// TwinCAT 3 PLC project PulsePower_PLC
// ProgramVersion: 3.1.4023.0
// libraries:
//   Tc2_BACnetRev12, * (Beckhoff Automation GmbH)
//   Tc2_DataExchange, * (Beckhoff Automation GmbH)
//   Tc2_Math, * (Beckhoff Automation GmbH)
//   Tc2_NC, * (Beckhoff Automation GmbH)
//   Tc2_Standard, * (Beckhoff Automation GmbH)
//   Tc2_System, * (Beckhoff Automation GmbH)
//   Tc3_EventLogger, * (Beckhoff Automation GmbH)
//   Tc3_Module, * (Beckhoff Automation GmbH)
// project tree:
//   DUTs/ E_Command.TcDUT, E_PulseState.TcDUT, E_Status.TcDUT, ST_Alarm_Base.TcDUT (not stored), ST_Charger_Base.TcDUT, ST_ChargeTime.TcDUT (not stored), ST_Control.TcDUT, ST_Echo_MCP.TcDUT, ST_Echo_Section.TcDUT, ST_FieldDevices_Base.TcDUT, ST_FieldDevices_Form.TcDUT (not stored), ST_InstrumentReading.TcDUT, ST_Recipe.TcDUT, ST_RelayFaults_Base.TcDUT (not stored), ST_RelayFaults_Form.TcDUT (not stored), ST_Section_Base.TcDUT (not stored), ST_Setpoints_Base.TcDUT (not stored), ST_Trip_Base.TcDUT (not stored), ST_VoltageFeedback.TcDUT (not stored)
//   GVLs/ Alarms_DB.TcGVL, ChargeTime_DB.TcGVL (not stored), Command.TcGVL (not stored), EngVal.TcGVL, GVL.TcGVL (not stored), Recipe.TcGVL, Setpoints.TcGVL, TxMainPLC.TcGVL, HMI_DB.TcGVL, Input.TcGVL, InstrumentReading.TcGVL, LCP.TcGVL (not stored), MCP_IO.TcGVL, Output.TcGVL, Permissives_DB.TcGVL, Trips_DB.TcGVL
//   / PlcTask.TcTTO
//   POUs/ ADC_10V.TcPOU (not stored), ADC_5V.TcPOU (not stored), Alarms.TcPOU, Alarms_FB.TcPOU (not stored), Alias.TcPOU, AnalogConversion.TcPOU, AQ.TcPOU (not stored), ChargeTime.TcPOU, Communication.TcPOU, Dump_FB.TcPOU, Heartbeat.TcPOU (not stored), Heartbeat_1.TcPOU, HMI.TcPOU, LCA_CAL.TcPOU (not stored), MAIN.TcPOU, Norm_x.TcPOU (not stored), Permissives.TcPOU, PWMO.TcPOU (not stored), Sequence.TcPOU, Trips.TcPOU
// real-time tasks:
//   TASK PlcTask: cycle T#2ms, priority 20, ADS port 350
// I/O:
//   DEVICE Device 3 (EtherCAT) (disabled), AmsNetId 5.107.141.148.4.1
//     Term 23 (EK1101) [EK1101 EtherCAT Coupler (2A E-Bus, ID switch)]
//       Term 24 (EL2008) [EL2008 8Ch. Dig. Output 24V, 0.5A]
//       Term 25 (EL2008) [EL2008 8Ch. Dig. Output 24V, 0.5A]
//       Term 26 (EL3068) [EL3068 8Ch. Ana. Input 0-10V]
//       Term 27 (EL3068) [EL3068 8Ch. Ana. Input 0-10V]
//       Term 28 (EL4008) [EL4008 8K. Ana. Ausgang 0-10V, 12bit]
//       Term 29 (EL2008) [EL2008 8Ch. Dig. Output 24V, 0.5A]
//       Term 30 (EL4008) [EL4008 8K. Ana. Ausgang 0-10V, 12bit]
//       Term 18 (EL9011) [EL9011 End Terminal]
//   DEVICE Device 2 (EtherCAT) (disabled), AmsNetId 5.107.141.148.3.1
//     Term 4 (EK1200) [EK1200-5000 EtherCAT Power supply (2A E-Bus)]
//       Term 2 (EL1008) [EL1008 8Ch. Dig. Input 24V, 3ms]
//       Term 3 (EL1008) [EL1008 8Ch. Dig. Input 24V, 3ms]
//       Term 4 (EL1008) [EL1008 8Ch. Dig. Input 24V, 3ms]
//       Term 5 (EL1008) [EL1008 8Ch. Dig. Input 24V, 3ms]
//       Term 6 (EL1008) [EL1008 8Ch. Dig. Input 24V, 3ms]
//       Term 7 (EL1008) [EL1008 8Ch. Dig. Input 24V, 3ms]
//       Term 11 (EL1008) [EL1008 8Ch. Dig. Input 24V, 3ms]
//       Term 12 (EL1008) [EL1008 8Ch. Dig. Input 24V, 3ms]
//       Term 13 (EL1008) [EL1008 8Ch. Dig. Input 24V, 3ms]
//       Term 14 (EL6695) [EL6695 EtherCAT Bridge terminal (Primary)]
//       Term 15 (EK1561) [EK1561 1 port EtherCAT junction (POF)]
//       Term 16 (EL9011) [EL9011 End Terminal]
// variable links:
//   PulsePower_PLC/PulsePower_PLC Instance <-> Device 2 (EtherCAT)/Term 4 (EK1200)/Term 11 (EL1008)
//     PlcTask Inputs/Input.R1_07_00 <-> Channel 1/Input
//     PlcTask Inputs/Input.R1_07_01 <-> Channel 2/Input
//     PlcTask Inputs/Input.R1_07_02 <-> Channel 3/Input
//     PlcTask Inputs/Input.R1_07_03 <-> Channel 4/Input
//     PlcTask Inputs/Input.R1_07_04 <-> Channel 5/Input
//     PlcTask Inputs/Input.R1_07_05 <-> Channel 6/Input
//     PlcTask Inputs/Input.R1_07_06 <-> Channel 7/Input
//     PlcTask Inputs/Input.R1_07_07 <-> Channel 8/Input
//   PulsePower_PLC/PulsePower_PLC Instance <-> Device 2 (EtherCAT)/Term 4 (EK1200)/Term 12 (EL1008)
//     PlcTask Inputs/Input.R1_08_00 <-> Channel 1/Input
//     PlcTask Inputs/Input.R1_08_01 <-> Channel 2/Input
//     PlcTask Inputs/Input.R1_08_02 <-> Channel 3/Input
//     PlcTask Inputs/Input.R1_08_03 <-> Channel 4/Input
//     PlcTask Inputs/Input.R1_08_04 <-> Channel 5/Input
//     PlcTask Inputs/Input.R1_08_05 <-> Channel 6/Input
//     PlcTask Inputs/Input.R1_08_06 <-> Channel 7/Input
//     PlcTask Inputs/Input.R1_08_07 <-> Channel 8/Input
//   PulsePower_PLC/PulsePower_PLC Instance <-> Device 2 (EtherCAT)/Term 4 (EK1200)/Term 13 (EL1008)
//     PlcTask Inputs/Input.R1_09_00 <-> Channel 1/Input
//     PlcTask Inputs/Input.R1_09_01 <-> Channel 2/Input
//     PlcTask Inputs/Input.R1_09_02 <-> Channel 3/Input
//     PlcTask Inputs/Input.R1_09_03 <-> Channel 4/Input
//     PlcTask Inputs/Input.R1_09_04 <-> Channel 5/Input
//     PlcTask Inputs/Input.R1_09_05 <-> Channel 6/Input
//     PlcTask Inputs/Input.R1_09_06 <-> Channel 7/Input
//     PlcTask Inputs/Input.R1_09_07 <-> Channel 8/Input
//   PulsePower_PLC/PulsePower_PLC Instance <-> Device 2 (EtherCAT)/Term 4 (EK1200)/Term 2 (EL1008)
//     PlcTask Inputs/Input.R1_01_00 <-> Channel 1/Input
//     PlcTask Inputs/Input.R1_01_01 <-> Channel 2/Input
//     PlcTask Inputs/Input.R1_01_02 <-> Channel 3/Input
//     PlcTask Inputs/Input.R1_01_03 <-> Channel 4/Input
//     PlcTask Inputs/Input.R1_01_04 <-> Channel 5/Input
//     PlcTask Inputs/Input.R1_01_05 <-> Channel 6/Input
//     PlcTask Inputs/Input.R1_01_06 <-> Channel 7/Input
//     PlcTask Inputs/Input.R1_01_07 <-> Channel 8/Input
//   PulsePower_PLC/PulsePower_PLC Instance <-> Device 2 (EtherCAT)/Term 4 (EK1200)/Term 3 (EL1008)
//     PlcTask Inputs/Input.R1_02_00 <-> Channel 1/Input
//     PlcTask Inputs/Input.R1_02_01 <-> Channel 2/Input
//     PlcTask Inputs/Input.R1_02_02 <-> Channel 3/Input
//     PlcTask Inputs/Input.R1_02_03 <-> Channel 4/Input
//     PlcTask Inputs/Input.R1_02_04 <-> Channel 5/Input
//     PlcTask Inputs/Input.R1_02_05 <-> Channel 6/Input
//     PlcTask Inputs/Input.R1_02_06 <-> Channel 7/Input
//     PlcTask Inputs/Input.R1_02_07 <-> Channel 8/Input
//   PulsePower_PLC/PulsePower_PLC Instance <-> Device 2 (EtherCAT)/Term 4 (EK1200)/Term 4 (EL1008)
//     PlcTask Inputs/Input.R1_03_00 <-> Channel 1/Input
//     PlcTask Inputs/Input.R1_03_01 <-> Channel 2/Input
//     PlcTask Inputs/Input.R1_03_02 <-> Channel 3/Input
//     PlcTask Inputs/Input.R1_03_03 <-> Channel 4/Input
//     PlcTask Inputs/Input.R1_03_04 <-> Channel 5/Input
//     PlcTask Inputs/Input.R1_03_05 <-> Channel 6/Input
//     PlcTask Inputs/Input.R1_03_06 <-> Channel 7/Input
//     PlcTask Inputs/Input.R1_03_07 <-> Channel 8/Input
//   PulsePower_PLC/PulsePower_PLC Instance <-> Device 2 (EtherCAT)/Term 4 (EK1200)/Term 5 (EL1008)
//     PlcTask Inputs/Input.R1_04_00 <-> Channel 1/Input
//     PlcTask Inputs/Input.R1_04_01 <-> Channel 2/Input
//     PlcTask Inputs/Input.R1_04_02 <-> Channel 3/Input
//     PlcTask Inputs/Input.R1_04_03 <-> Channel 4/Input
//     PlcTask Inputs/Input.R1_04_04 <-> Channel 5/Input
//     PlcTask Inputs/Input.R1_04_05 <-> Channel 6/Input
//     PlcTask Inputs/Input.R1_04_06 <-> Channel 7/Input
//     PlcTask Inputs/Input.R1_04_07 <-> Channel 8/Input
//   PulsePower_PLC/PulsePower_PLC Instance <-> Device 2 (EtherCAT)/Term 4 (EK1200)/Term 6 (EL1008)
//     PlcTask Inputs/Input.R1_05_00 <-> Channel 1/Input
//     PlcTask Inputs/Input.R1_05_01 <-> Channel 2/Input
//     PlcTask Inputs/Input.R1_05_02 <-> Channel 3/Input
//     PlcTask Inputs/Input.R1_05_03 <-> Channel 4/Input
//     PlcTask Inputs/Input.R1_05_04 <-> Channel 5/Input
//     PlcTask Inputs/Input.R1_05_05 <-> Channel 6/Input
//     PlcTask Inputs/Input.R1_05_06 <-> Channel 7/Input
//     PlcTask Inputs/Input.R1_05_07 <-> Channel 8/Input
//   PulsePower_PLC/PulsePower_PLC Instance <-> Device 2 (EtherCAT)/Term 4 (EK1200)/Term 7 (EL1008)
//     PlcTask Inputs/Input.R1_06_00 <-> Channel 1/Input
//     PlcTask Inputs/Input.R1_06_01 <-> Channel 2/Input
//     PlcTask Inputs/Input.R1_06_02 <-> Channel 3/Input
//     PlcTask Inputs/Input.R1_06_03 <-> Channel 4/Input
//     PlcTask Inputs/Input.R1_06_04 <-> Channel 5/Input
//     PlcTask Inputs/Input.R1_06_05 <-> Channel 6/Input
//     PlcTask Inputs/Input.R1_06_06 <-> Channel 7/Input
//     PlcTask Inputs/Input.R1_06_07 <-> Channel 8/Input
//   PulsePower_PLC/PulsePower_PLC Instance <-> Device 3 (EtherCAT)/Term 23 (EK1101)/Term 24 (EL2008)
//     PlcTask Outputs/Output.R2_01_00 <-> Channel 1/Output
//     PlcTask Outputs/Output.R2_01_01 <-> Channel 2/Output
//     PlcTask Outputs/Output.R2_01_02 <-> Channel 3/Output
//     PlcTask Outputs/Output.R2_01_03 <-> Channel 4/Output
//     PlcTask Outputs/Output.R2_01_04 <-> Channel 5/Output
//     PlcTask Outputs/Output.R2_01_05 <-> Channel 6/Output
//     PlcTask Outputs/Output.R2_01_06 <-> Channel 7/Output
//     PlcTask Outputs/Output.R2_01_07 <-> Channel 8/Output
//   PulsePower_PLC/PulsePower_PLC Instance <-> Device 3 (EtherCAT)/Term 23 (EK1101)/Term 25 (EL2008)
//     PlcTask Outputs/Output.R2_02_00 <-> Channel 1/Output
//     PlcTask Outputs/Output.R2_02_01 <-> Channel 2/Output
//     PlcTask Outputs/Output.R2_02_02 <-> Channel 3/Output
//     PlcTask Outputs/Output.R2_02_03 <-> Channel 4/Output
//     PlcTask Outputs/Output.R2_02_04 <-> Channel 5/Output
//     PlcTask Outputs/Output.R2_02_05 <-> Channel 6/Output
//     PlcTask Outputs/Output.R2_02_06 <-> Channel 7/Output
//     PlcTask Outputs/Output.R2_02_07 <-> Channel 8/Output
//   PulsePower_PLC/PulsePower_PLC Instance <-> Device 3 (EtherCAT)/Term 23 (EK1101)/Term 26 (EL3068)
//     PlcTask Inputs/Input.R2_03_00 <-> AI Standard Channel 1/Value
//     PlcTask Inputs/Input.R2_03_01 <-> AI Standard Channel 2/Value
//     PlcTask Inputs/Input.R2_03_02 <-> AI Standard Channel 3/Value
//     PlcTask Inputs/Input.R2_03_03 <-> AI Standard Channel 4/Value
//     PlcTask Inputs/Input.R2_03_04 <-> AI Standard Channel 5/Value
//     PlcTask Inputs/Input.R2_03_05 <-> AI Standard Channel 6/Value
//     PlcTask Inputs/Input.R2_03_06 <-> AI Standard Channel 7/Value
//     PlcTask Inputs/Input.R2_03_07 <-> AI Standard Channel 8/Value
//     PlcTask Inputs/Input.R2_03_00_Status <-> AI Standard Channel 1/Status
//     PlcTask Inputs/Input.R2_03_01_Status <-> AI Standard Channel 2/Status
//     PlcTask Inputs/Input.R2_03_02_Status <-> AI Standard Channel 3/Status
//     PlcTask Inputs/Input.R2_03_03_Status <-> AI Standard Channel 4/Status
//     PlcTask Inputs/Input.R2_03_04_Status <-> AI Standard Channel 5/Status
//     PlcTask Inputs/Input.R2_03_05_Status <-> AI Standard Channel 6/Status
//     PlcTask Inputs/Input.R2_03_06_Status <-> AI Standard Channel 7/Status
//     PlcTask Inputs/Input.R2_03_07_Status <-> AI Standard Channel 8/Status
//   PulsePower_PLC/PulsePower_PLC Instance <-> Device 3 (EtherCAT)/Term 23 (EK1101)/Term 27 (EL3068)
//     PlcTask Inputs/Input.R2_04_00 <-> AI Standard Channel 1/Value
//     PlcTask Inputs/Input.R2_04_01 <-> AI Standard Channel 2/Value
//     PlcTask Inputs/Input.R2_04_02 <-> AI Standard Channel 3/Value
//     PlcTask Inputs/Input.R2_04_03 <-> AI Standard Channel 4/Value
//     PlcTask Inputs/Input.R2_04_04 <-> AI Standard Channel 5/Value
//     PlcTask Inputs/Input.R2_04_05 <-> AI Standard Channel 6/Value
//     PlcTask Inputs/Input.R2_04_06 <-> AI Standard Channel 7/Value
//     PlcTask Inputs/Input.R2_04_07 <-> AI Standard Channel 8/Value
//     PlcTask Inputs/Input.R2_04_00_Status <-> AI Standard Channel 1/Status
//     PlcTask Inputs/Input.R2_04_01_Status <-> AI Standard Channel 2/Status
//     PlcTask Inputs/Input.R2_04_02_Status <-> AI Standard Channel 3/Status
//     PlcTask Inputs/Input.R2_04_03_Status <-> AI Standard Channel 4/Status
//     PlcTask Inputs/Input.R2_04_04_Status <-> AI Standard Channel 5/Status
//     PlcTask Inputs/Input.R2_04_05_Status <-> AI Standard Channel 6/Status
//     PlcTask Inputs/Input.R2_04_06_Status <-> AI Standard Channel 7/Status
//     PlcTask Inputs/Input.R2_04_07_Status <-> AI Standard Channel 8/Status
//   PulsePower_PLC/PulsePower_PLC Instance <-> Device 3 (EtherCAT)/Term 23 (EK1101)/Term 28 (EL4008)
//     PlcTask Outputs/Output.R2_05_00 <-> AO Outputs Channel 1/Analog output
//     PlcTask Outputs/Output.R2_05_01 <-> AO Outputs Channel 2/Analog output
//     PlcTask Outputs/Output.R2_05_02 <-> AO Outputs Channel 3/Analog output
//     PlcTask Outputs/Output.R2_05_03 <-> AO Outputs Channel 4/Analog output
//     PlcTask Outputs/Output.R2_05_04 <-> AO Outputs Channel 5/Analog output
//     PlcTask Outputs/Output.R2_05_05 <-> AO Outputs Channel 6/Analog output
//     PlcTask Outputs/Output.R2_05_06 <-> AO Outputs Channel 7/Analog output
//     PlcTask Outputs/Output.R2_05_07 <-> AO Outputs Channel 8/Analog output
//   PulsePower_PLC/PulsePower_PLC Instance <-> Device 3 (EtherCAT)/Term 23 (EK1101)/Term 29 (EL2008)
//     PlcTask Outputs/Output.R2_06_00 <-> Channel 1/Output
//     PlcTask Outputs/Output.R2_06_01 <-> Channel 2/Output
//     PlcTask Outputs/Output.R2_06_02 <-> Channel 3/Output
//     PlcTask Outputs/Output.R2_06_03 <-> Channel 4/Output
//     PlcTask Outputs/Output.R2_06_04 <-> Channel 5/Output
//     PlcTask Outputs/Output.R2_06_05 <-> Channel 6/Output
//     PlcTask Outputs/Output.R2_06_06 <-> Channel 7/Output
//     PlcTask Outputs/Output.R2_06_07 <-> Channel 8/Output
//   PulsePower_PLC/PulsePower_PLC Instance <-> Device 3 (EtherCAT)/Term 23 (EK1101)/Term 30 (EL4008)
//     PlcTask Outputs/Output.R2_07_00 <-> AO Outputs Channel 1/Analog output
//     PlcTask Outputs/Output.R2_07_01 <-> AO Outputs Channel 2/Analog output
//     PlcTask Outputs/Output.R2_07_02 <-> AO Outputs Channel 3/Analog output
//     PlcTask Outputs/Output.R2_07_03 <-> AO Outputs Channel 4/Analog output
//     PlcTask Outputs/Output.R2_07_04 <-> AO Outputs Channel 5/Analog output
//     PlcTask Outputs/Output.R2_07_05 <-> AO Outputs Channel 6/Analog output
//     PlcTask Outputs/Output.R2_07_06 <-> AO Outputs Channel 7/Analog output
//     PlcTask Outputs/Output.R2_07_07 <-> AO Outputs Channel 8/Analog output

CONFIGURATION PulsePower_PLC
    RESOURCE PLC ON TwinCAT3
        TASK PlcTask(INTERVAL := T#2ms, PRIORITY := 20);
        PROGRAM MAIN WITH PlcTask : MAIN;
        PROGRAM Heartbeat WITH PlcTask : Heartbeat;
        PROGRAM Heartbeat_1 WITH PlcTask : Heartbeat_1;
    END_RESOURCE
END_CONFIGURATION

// ---- DUTs/E_Command.TcDUT
{attribute 'qualified_only'}
{attribute 'strict'}
{attribute 'to_string'}
//Command from Master PLC (screenroom)
TYPE E_Command :
(
	//Requested PP State
	IDLE		 	:= 0, 
	CHARGE			:= 1, 
	DISCONNECT		:= 2,
	DUMP			:= 3, 
	ABORT			:= 4
);
END_TYPE

// ---- DUTs/E_PulseState.TcDUT
{attribute 'qualified_only'}
{attribute 'strict'}
TYPE E_PulseState :
(
	SAFE			:= 0, //IDLE
	CHARGING		:= 1, //Charge
	CHARGECOMPLETE	:= 2, //EOC
	DISCONNECTING	:= 3, //Disconnect
	DUMPING			:= 4, 
	ABORT			:= 5,
	TRIPPED			:= 6,
	LOCALMODE		:= 7	
);
END_TYPE

// ---- DUTs/E_Status.TcDUT
{attribute 'qualified_only'}
{attribute 'strict'}
{attribute 'to_string'}
TYPE E_Status :
(
	//Actual Pulse Power State
	SAFE			:= 0, //IDLE
	CHARGING		:= 1, //Charge
	CHARGECOMPLETE	:= 2, //EOC
	DISCONNECTING	:= 3, //Disconnect
	DISCONNECTED	:= 4,
	DUMPING			:= 5, 
	ABORT			:= 6,	
	TRIPPED			:= 7,
	LOCAL_MODE		:= 8
) ;
END_TYPE

// ---- DUTs/ST_Charger_Base.TcDUT
TYPE ST_Charger_Base :
STRUCT
	//DI
	inhibited 		: BOOL;
	EndOfCharge 	: BOOL;
	HV_isON			: BOOL;
	OverTemp		: BOOL;
	InterlockOpen	: BOOL;
	LoadFaulted		: BOOL;
	SummaryFaulted	: BOOL;
	
	//DQ
	inhibit			: BOOL;
	HV_ON			: BOOL;
	
	//AI
	voltageFeedback_raw 	: INT;
	voltageFeedback_norm 	: REAL;
	voltageFeedback			: REAL;
	
	currentFeedback_raw 	: INT;
	currentFeedback_norm	: REAL;
	currentFeedback			: REAL;
	
	//AQ
	voltageSP_norm	: REAL;
	voltageSP		: DINT;
	voltageSP_raw	: INT; // setpoint output to field device.
	
	//Internal
	ChargerType_50kV : BOOL;
	ChargerType_12kV : BOOL;
	LossInhibit		 : BOOL;
	LossHVON		 : BOOL;
	LossInhibitTON	 : TON;
	LossHVON_TON	 : TON;
	
	ChargeTime		: ST_ChargeTime;
END_STRUCT
END_TYPE

// ---- DUTs/ST_Control.TcDUT
TYPE ST_Control :
STRUCT
	ClearAllFaults : BOOL;
END_STRUCT
END_TYPE

// ---- DUTs/ST_Echo_MCP.TcDUT
TYPE ST_Echo_MCP :
STRUCT
	VoltageFeedback : REAL;
	CurrentFeedback : REAL;
	TDKLoad			: ST_ChargeTime;
	
END_STRUCT
END_TYPE

// ---- DUTs/ST_Echo_Section.TcDUT
TYPE ST_Echo_Section :
STRUCT
	PeakCap : ARRAY[1..10] OF ST_InstrumentReading;
	SustCap : ARRAY[1..2] OF ST_InstrumentReading;
	FormCap : ARRAY[1..12] OF ST_InstrumentReading;
	FormTrigVoltage		: REAL;
	PreFormTrigVoltage  : REAL;
	PreFormCapVoltage  : REAL;
END_STRUCT
END_TYPE

// ---- DUTs/ST_FieldDevices_Base.TcDUT
TYPE ST_FieldDevices_Base :
STRUCT
	Cap : ARRAY [1..12] OF ST_InstrumentReading;
	
	ChargeRelay1_close		:BOOL;
	ChargeRelay2_close		:BOOL;
	
	ShortContact1_close		:BOOL;
	UnshortContact1_close 	:BOOL;
	ShortContact1Engaged	:BOOL;
	ShortContact1unknown	:BOOL;
	
	ShortContact2_close		:BOOL;
	UnshortContact2_close 	:BOOL;
	ShortContact2Engaged	:BOOL;
	ShortContact2unknown	:BOOL;
	
	DumpRelay1_close		:BOOL;
	DumpRelay2_close		:BOOL;
	
	CloseChargeRelay1		:BOOL;
	CloseChargeRelay2		:BOOL;
	OpenDumpRelay1			:BOOL;
	OpenDumpRelay2			:BOOL;
	
	//Bank					: ST_ChargeTime;

END_STRUCT
END_TYPE

// ---- DUTs/ST_InstrumentReading.TcDUT
TYPE ST_InstrumentReading :
STRUCT
	
	(*CH00 : REAL;
	CH01 : REAL;
	CH02 : REAL;
	CH03 : REAL;
	CH04 : REAL;
	CH05 : REAL;
	CH06 : REAL;
	CH07 : REAL;
	R2_01_CH02 : REAL;
	R2_01_CH03 : REAL;
	R2_01_CH04 : REAL;
	R2_01_CH05 : REAL;
	R2_01_CH06 : REAL;
	R2_01_CH07 : REAL;*)
	voltageFeedback_raw		: INT;
	voltageFeedback_Norm 	: REAL;
	voltageFeedback 		: REAL;
	currentFeedback_raw		: INT;
	currentFeedback_Norm 	: REAL;
	currentFeedback 		: REAL;
	
	CapDischaged			: BOOL;
	CapFullyCharged			: BOOL;
END_STRUCT
END_TYPE

// ---- DUTs/ST_Recipe.TcDUT
TYPE ST_Recipe :
STRUCT
	RequiredChargedV : REAL := 10; //DINT;
END_STRUCT
END_TYPE

// ---- GVLs/Alarms_DB.TcGVL
{attribute 'qualified_only'}
VAR_GLOBAL
	MCP	: ST_Alarm_Base;
	Section1 : ST_Alarm_Base;
	Section2 : ST_Alarm_Base;
	Section3 : ST_Alarm_Base;
	Section4 : ST_Alarm_Base;
	
	AlarmWord5  : ST_Alarm_Base;
	AlarmWord6  : ST_Alarm_Base;
	AlarmWord7  : ST_Alarm_Base;
	AlarmWord8  : ST_Alarm_Base;
	AlarmWord9  : ST_Alarm_Base;
	//AlarmWord11 : ST_Alarm_Base;
	//AlarmWord12 : ST_Alarm_Base;
	//AlarmWord13 : ST_Alarm_Base;
	//AlarmWord14 : ST_Alarm_Base;
	//AlarmWord15 : ST_Alarm_Base;
END_VAR

// ---- GVLs/EngVal.TcGVL
{attribute 'qualified_only'}
VAR_GLOBAL
	Max_50kVChargerVoltage : REAL := 50000; //50kV
	Min_50kVChargerVoltage : REAL := 0;
	
	Max_50kVChargerCurrent : REAL := 0.18; //total peak charge current is 0.18A
	Min_50kVChargerCurrent : REAL := 0;
	
	Max_12kVChargerVoltage : REAL := 12000; //12kV
	Min_12kVChargerVoltage : REAL := 0;
	
	Max_12kVChargerCurrent : REAL := 0.75; //total peak charge current is 0.75A
	Min_12kVChargerCurrent : REAL := 0;
	
	Max_GLS1_ChargerV	   : REAL := 50000; //form trigger
	Max_GLS2_ChargerV	   : REAL := 50000; // preform trigger
	Max_GLS3_ChargerV	   : REAL := 30000; // preform cap charger
	
	Max_CapVoltage			: REAL := 32000;  //assuming 32kV cap....  
	Min_CapVoltage			: REAL := 0;
	
	ULimit_PeakCapRequiredV	: REAL := 10000; //10kV veto
	LLimit_PeakCapRequiredV	: REAL := -2000; //-2kV
	ULimit_SustCapRequiredV	: REAL := 12000; //12kv veto
	LLimit_SustCapRequiredV	: REAL := -2000; //-2kv
	ULimit_FormCapRequiredV : REAL := 35000;
	LLimit_FormCapRequiredV : REAL := 0;
	
	ULimit_PreFormCapRequiredV : REAL := 30000;
	LLimit_PreFormCapRequiredV : REAL := 0;
		
END_VAR

// ---- GVLs/Recipe.TcGVL
{attribute 'qualified_only'}
VAR_GLOBAL
	TDKLoad : ARRAY [1..8] OF ST_Recipe;
	GLSLoad : ST_Recipe;
	GLS1_VSP : REAL := 50; //DINT;
	GLS2_VSP : REAL := 50; //DINT;
END_VAR

// ---- GVLs/Setpoints.TcGVL
{attribute 'qualified_only'}
VAR_GLOBAL
	TDKLoad : ARRAY [1..8] OF ST_Setpoints_Base;
	GLSLoad : ST_Setpoints_Base;
	GLS1_VSP : REAL := 50;
	GLS2_VSP : REAL := 50;
END_VAR

// ---- GVLs/TxMainPLC.TcGVL
{attribute 'qualified_only'}
VAR_GLOBAL
	Charger		: ARRAY[1..8] OF ST_Echo_MCP;
	GLSLoad		: ST_ChargeTime;
	Section 	: ARRAY[1..4] OF ST_Echo_Section;
	ChargeRunOutTime	: REAL;
	ChargingRunOutTime	: REAL;
END_VAR

// ---- GVLs/HMI_DB.TcGVL
{attribute 'qualified_only'}
VAR_GLOBAL PERSISTENT
	RemoteModeSelected 	: BOOL := TRUE;
	
	OpenAllDumpRlyPB	: BOOL;
	CloseAllChargeRlyPB	: BOOL;
	AbortPB				: BOOL;
	
	ChargerHVOFF_rlyDelayPT		: TIME := T#25MS;
	ChargerHVOFF_rlyDelayPT_INT	: INT := 25;
	
	HVONdelayPT					: TIME := T#250MS;
	HVONdelayPT_INT				: INT := 250;
	
	RunOutTMR_PT				: TIME := T#10S;
	RunOutTMR_PT_INT			: INT := 10;
	RunOutTMR_elapse			: INT;
	
	ChargingRunOutTMR_elapse	: INT;
	
	//admin bypasses
	SafetyOKBP					: BOOL;
	AllDumpRelaysOpenBP			: BOOL;
	InterlockPressureLossBP		: BOOL;
	AllChargeRelayCloseBP		: BOOL;
	NoFaultDetectedBP			: BOOL;
	//AllShortingSysRemovedBP		: BOOL;
	AlldcPSUokBP				: BOOL;
	LossHVsignalBP				: BOOL;
	
	//timeToChargeLoad 			: ARRAY [1..8] OF REAL;
	//GLSchargeTime	 			: ARRAY [1..3] OF REAL;
	TDKLoad 					: ARRAY [1..8] OF ST_Setpoints_Base; //or RETAIN
	GLSLoad	 					: ST_Setpoints_Base;
	
	(*PSratedV					: REAL := 50;
	RequiredChargeV				: REAL := 30;
	LoadCapacitance				: REAL := 600;
	wLCA						: BOOL := TRUE;
	NumOfCharger				: INT := 1;*)
END_VAR

VAR_GLOBAL
	LiftMachineGNDsw			: BOOL;
	//for startup run
	PeakChargerSP				: DINT;
	SustChargerSP				: DINT;
	FormChargerSP				: DINT;
	PreFormChargerSP			: DINT;
	FormTrigChargerSP			: DINT;
	PreFormTrigChargerSP		: DINT;
	
	OpenAllPeakDumpRlySW		: BOOL;
	OpenAllSustDumpRlySW		: BOOL;
	OpenAllFormDumpRlySW		: BOOL;
	OpenAllPreFormDumpRlySW		: BOOL;
	OpenFormTrigDumpRlySW		: BOOL;
	OpenPreFormTrigDumpRlySW	: BOOL;
	
	CloseAllPeakChargRlySW		: BOOL;
	CloseAllSustChargRlySW		: BOOL;
	CloseAllFormChargRlySW		: BOOL;
	CloseAllPreFormChargRlySW	: BOOL;
	CloseFormTrigChargeRlySW	: BOOL;
	ClosePreFormTrigChargeRlySW : BOOL;
	
	PeakHVONsw					: BOOL; //enable
	SustHVONsw					: BOOL; //enable
	FormHVONsw					: BOOL; //enable
	PreFormHVONsw				: BOOL;
	GLS1HVONsw					: BOOL;
	GLS2HVONsw					: BOOL;
	
	ResetPB_Local				: BOOL;
	
	(*PeakInhibitONsw				: BOOL;
	SustInhibitONsw				: BOOL;
	FormInhibitONsw				: BOOL;
	PreFormInhibitONsw			: BOOL;
	*)	
END_VAR

// ---- GVLs/Input.TcGVL
{attribute 'qualified_only'}
VAR_GLOBAL
//***MCP************************************************************************
	//EL1008 - DI1
	R1_01_00 AT	%I*: BOOL; //Master stop PB not pressed - black pb on mcp
	R1_01_01 AT	%I*: BOOL; //case Estop circuit okay (Rly1 (120vac)
	R1_01_02 AT %I*: BOOL; //Remote Mode Selected (NO)
	R1_01_03 AT %I*: BOOL; //MCP PSU1 DC OK
	R1_01_04 AT %I*: BOOL; //Machine Ground Relay Open (lifted) Opto Board
	R1_01_05 AT %I*: BOOL; //spare
	R1_01_06 AT %I*: BOOL; //spare
	R1_01_07 AT %I*: BOOL; //spare

	//EL1008 - DI2
	//TDK802 1
	R1_02_00 AT	%I*: BOOL; 
	R1_02_01 AT	%I*: BOOL;
	R1_02_02 AT %I*: BOOL; 
	R1_02_03 AT %I*: BOOL; 
	R1_02_04 AT %I*: BOOL; 
	R1_02_05 AT %I*: BOOL; 
	R1_02_06 AT %I*: BOOL; 
	R1_02_07 AT %I*: BOOL; //spare
	
	//EL1008 - DI3
	//TDK802 2
	R1_03_00 AT	%I*: BOOL; 
	R1_03_01 AT	%I*: BOOL;
	R1_03_02 AT %I*: BOOL; 
	R1_03_03 AT %I*: BOOL; 
	R1_03_04 AT %I*: BOOL; 
	R1_03_05 AT %I*: BOOL; 
	R1_03_06 AT %I*: BOOL; 
	R1_03_07 AT %I*: BOOL; //spare
		
	//EL1008 - DI4
	//TDK802 3
	R1_04_00 AT	%I*: BOOL; 
	R1_04_01 AT	%I*: BOOL;
	R1_04_02 AT %I*: BOOL; 
	R1_04_03 AT %I*: BOOL; 
	R1_04_04 AT %I*: BOOL; 
	R1_04_05 AT %I*: BOOL; 
	R1_04_06 AT %I*: BOOL; 
	R1_04_07 AT %I*: BOOL; //spare
	
	//EL1008 - DI5
	//TDK802 4
	R1_05_00 AT	%I*: BOOL; 
	R1_05_01 AT	%I*: BOOL;
	R1_05_02 AT %I*: BOOL; 
	R1_05_03 AT %I*: BOOL; 
	R1_05_04 AT %I*: BOOL; 
	R1_05_05 AT %I*: BOOL; 
	R1_05_06 AT %I*: BOOL; 
	R1_05_07 AT %I*: BOOL; //spare
	
	//EL1008 - DI6
	//TDK802 5
	R1_06_00 AT	%I*: BOOL; 
	R1_06_01 AT	%I*: BOOL;
	R1_06_02 AT %I*: BOOL; 
	R1_06_03 AT %I*: BOOL; 
	R1_06_04 AT %I*: BOOL; 
	R1_06_05 AT %I*: BOOL; 
	R1_06_06 AT %I*: BOOL; 
	R1_06_07 AT %I*: BOOL; //spare
	
	//EL1008 - DI7
	//TDK802 6
	R1_07_00 AT	%I*: BOOL; 
	R1_07_01 AT	%I*: BOOL;
	R1_07_02 AT %I*: BOOL; 
	R1_07_03 AT %I*: BOOL; 
	R1_07_04 AT %I*: BOOL; 
	R1_07_05 AT %I*: BOOL; 
	R1_07_06 AT %I*: BOOL; 
	R1_07_07 AT %I*: BOOL; //spare
	
	//EL1008 - DI8
	//TDK802 7
	R1_08_00 AT	%I*: BOOL; 
	R1_08_01 AT	%I*: BOOL;
	R1_08_02 AT %I*: BOOL; 
	R1_08_03 AT %I*: BOOL; 
	R1_08_04 AT %I*: BOOL; 
	R1_08_05 AT %I*: BOOL; 
	R1_08_06 AT %I*: BOOL; 
	R1_08_07 AT %I*: BOOL; //spare
	
	//EL1008 - DI9
	//TDK802 8
	R1_09_00 AT	%I*: BOOL; 
	R1_09_01 AT	%I*: BOOL;
	R1_09_02 AT %I*: BOOL; 
	R1_09_03 AT %I*: BOOL; 
	R1_09_04 AT %I*: BOOL; 
	R1_09_05 AT %I*: BOOL; 
	R1_09_06 AT %I*: BOOL; 
	R1_09_07 AT %I*: BOOL; //spare

//RACK 2
	//EL3068 - AI1
	R2_03_00 		AT %I*: INT;
	R2_03_00_Status AT %I*: WORD;

	R2_03_01 		AT %I*: INT;
	R2_03_01_Status AT %I*: WORD;

	R2_03_02 		AT %I*: INT;
	R2_03_02_Status AT %I*: WORD;

	R2_03_03 		AT %I*: INT;
	R2_03_03_Status AT %I*: WORD;

	R2_03_04 		AT %I*: INT;
	R2_03_04_Status AT %I*: WORD;

	R2_03_05 		AT %I*: INT;
	R2_03_05_Status AT %I*: WORD;

	R2_03_06 		AT %I*: INT;
	R2_03_06_Status AT %I*: WORD;

	R2_03_07 		AT %I*: INT;
	R2_03_07_Status AT %I*: WORD;


	//EL3068 - AI2
	R2_04_00 		AT %I*: INT;
	R2_04_00_Status AT %I*: WORD;

	R2_04_01 		AT %I*: INT;
	R2_04_01_Status AT %I*: WORD;

	R2_04_02 		AT %I*: INT;
	R2_04_02_Status AT %I*: WORD;

	R2_04_03 		AT %I*: INT;
	R2_04_03_Status AT %I*: WORD;

	R2_04_04 		AT %I*: INT;
	R2_04_04_Status AT %I*: WORD;

	R2_04_05 		AT %I*: INT;
	R2_04_05_Status AT %I*: WORD;

	R2_04_06 		AT %I*: INT;
	R2_04_06_Status AT %I*: WORD;

	R2_04_07 		AT %I*: INT;
	R2_04_07_Status AT %I*: WORD;

//***LCP1***BANK1 (Rack 3)********************************************************************
//EL3068 - AI1
	R3_01_00 		AT %I*: INT;
	R3_01_00_Status AT %I*: WORD;
	
	R3_01_01		AT %I*: INT;
	R3_01_01_Status AT %I*: WORD;
	
	R3_01_02 		AT %I*: INT;
	R3_01_02_Status AT %I*: WORD;
	
	R3_01_03 		AT %I*: INT;
	R3_01_03_Status AT %I*: WORD;
	
	R3_01_04 		AT %I*: INT;
	R3_01_04_Status AT %I*: WORD;
	
	R3_01_05 		AT %I*: INT;
	R3_01_05_Status AT %I*: WORD;
	
	R3_01_06 		AT %I*: INT;
	R3_01_06_Status AT %I*: WORD;
	
	R3_01_07 		AT %I*: INT;
	R3_01_07_Status AT %I*: WORD;
	
	//EL3068 - AI2
	R3_02_00 		AT %I*: INT;
	R3_02_00_Status AT %I*: WORD;
	
	R3_02_01		AT %I*: INT;
	R3_02_01_Status AT %I*: WORD;
	
	R3_02_02 		AT %I*: INT;
	R3_02_02_Status AT %I*: WORD;
	
	R3_02_03 		AT %I*: INT;
	R3_02_03_Status AT %I*: WORD;
	
	R3_02_04 		AT %I*: INT; //SPARE
	R3_02_04_Status AT %I*: WORD;
	
	R3_02_05 		AT %I*: INT; //SPARE
	R3_02_05_Status AT %I*: WORD;
	
	R3_02_06 		AT %I*: INT; //SPARE
	R3_02_06_Status AT %I*: WORD;
	
	R3_02_07 		AT %I*: INT; //SPARE
	R3_02_07_Status AT %I*: WORD;

//EL1008 - DI1
	R3_03_00 AT %I*: BOOL;
	R3_03_01 AT %I*: BOOL;
	R3_03_02 AT %I*: BOOL;
	R3_03_03 AT %I*: BOOL;
	R3_03_04 AT %I*: BOOL;
	R3_03_05 AT %I*: BOOL;
	R3_03_06 AT %I*: BOOL;
	R3_03_07 AT %I*: BOOL;
//EL1008 - DI2	
	R3_04_00 AT %I*: BOOL;
	R3_04_01 AT %I*: BOOL;
	R3_04_02 AT %I*: BOOL;
	R3_04_03 AT %I*: BOOL;
	R3_04_04 AT %I*: BOOL;
	R3_04_05 AT %I*: BOOL; 
	R3_04_06 AT %I*: BOOL; //SPARE
	R3_04_07 AT %I*: BOOL; //SPARE

//***LCP2***BANK2 (Rack 4)********************************************************************
//EL3068 - AI1
	R4_01_00 		AT %I*: INT;
	R4_01_00_Status AT %I*: WORD;
	
	R4_01_01		AT %I*: INT;
	R4_01_01_Status AT %I*: WORD;
	
	R4_01_02 		AT %I*: INT;
	R4_01_02_Status AT %I*: WORD;
	
	R4_01_03 		AT %I*: INT;
	R4_01_03_Status AT %I*: WORD;
	
	R4_01_04 		AT %I*: INT;
	R4_01_04_Status AT %I*: WORD;
	
	R4_01_05 		AT %I*: INT;
	R4_01_05_Status AT %I*: WORD;
	
	R4_01_06 		AT %I*: INT;
	R4_01_06_Status AT %I*: WORD;
	
	R4_01_07 		AT %I*: INT;
	R4_01_07_Status AT %I*: WORD;
	
	//EL3068 - AI2
	R4_02_00 		AT %I*: INT;
	R4_02_00_Status AT %I*: WORD;
	
	R4_02_01		AT %I*: INT;
	R4_02_01_Status AT %I*: WORD;
	
	R4_02_02 		AT %I*: INT;
	R4_02_02_Status AT %I*: WORD;
	
	R4_02_03 		AT %I*: INT;
	R4_02_03_Status AT %I*: WORD;
	
	R4_02_04 		AT %I*: INT; //SPARE
	R4_02_04_Status AT %I*: WORD;
	
	R4_02_05 		AT %I*: INT; //SPARE
	R4_02_05_Status AT %I*: WORD;
	
	R4_02_06 		AT %I*: INT; //SPARE
	R4_02_06_Status AT %I*: WORD;
	
	R4_02_07 		AT %I*: INT; //SPARE
	R4_02_07_Status AT %I*: WORD;

//EL1008 - DI1
	R4_03_00 AT %I*: BOOL;
	R4_03_01 AT %I*: BOOL;
	R4_03_02 AT %I*: BOOL;
	R4_03_03 AT %I*: BOOL;
	R4_03_04 AT %I*: BOOL;
	R4_03_05 AT %I*: BOOL;
	R4_03_06 AT %I*: BOOL;
	R4_03_07 AT %I*: BOOL;
//EL1008 - DI2	
	R4_04_00 AT %I*: BOOL;
	R4_04_01 AT %I*: BOOL;
	R4_04_02 AT %I*: BOOL;
	R4_04_03 AT %I*: BOOL;
	R4_04_04 AT %I*: BOOL;
	R4_04_05 AT %I*: BOOL; 
	R4_04_06 AT %I*: BOOL; //SPARE
	R4_04_07 AT %I*: BOOL; //SPARE

//***LCP3***BANK3 (Rack 5)********************************************************************
//EL3068 - AI1
	R5_01_00 		AT %I*: INT;
	R5_01_00_Status AT %I*: WORD;
	
	R5_01_01		AT %I*: INT;
	R5_01_01_Status AT %I*: WORD;
	
	R5_01_02 		AT %I*: INT;
	R5_01_02_Status AT %I*: WORD;
	
	R5_01_03 		AT %I*: INT;
	R5_01_03_Status AT %I*: WORD;
	
	R5_01_04 		AT %I*: INT;
	R5_01_04_Status AT %I*: WORD;
	
	R5_01_05 		AT %I*: INT;
	R5_01_05_Status AT %I*: WORD;
	
	R5_01_06 		AT %I*: INT;
	R5_01_06_Status AT %I*: WORD;
	
	R5_01_07 		AT %I*: INT;
	R5_01_07_Status AT %I*: WORD;
	
	//EL3068 - AI2
	R5_02_00 		AT %I*: INT;
	R5_02_00_Status AT %I*: WORD;
	
	R5_02_01		AT %I*: INT;
	R5_02_01_Status AT %I*: WORD;
	
	R5_02_02 		AT %I*: INT;
	R5_02_02_Status AT %I*: WORD;
	
	R5_02_03 		AT %I*: INT;
	R5_02_03_Status AT %I*: WORD;
	
	R5_02_04 		AT %I*: INT; //SPARE
	R5_02_04_Status AT %I*: WORD;
	
	R5_02_05 		AT %I*: INT; //SPARE
	R5_02_05_Status AT %I*: WORD;
	
	R5_02_06 		AT %I*: INT; //SPARE
	R5_02_06_Status AT %I*: WORD;
	
	R5_02_07 		AT %I*: INT; //SPARE
	R5_02_07_Status AT %I*: WORD;

//EL1008 - DI1
	R5_03_00 AT %I*: BOOL;
	R5_03_01 AT %I*: BOOL;
	R5_03_02 AT %I*: BOOL;
	R5_03_03 AT %I*: BOOL;
	R5_03_04 AT %I*: BOOL;
	R5_03_05 AT %I*: BOOL;
	R5_03_06 AT %I*: BOOL;
	R5_03_07 AT %I*: BOOL;
//EL1008 - DI2	
	R5_04_00 AT %I*: BOOL;
	R5_04_01 AT %I*: BOOL;
	R5_04_02 AT %I*: BOOL;
	R5_04_03 AT %I*: BOOL;
	R5_04_04 AT %I*: BOOL;
	R5_04_05 AT %I*: BOOL; 
	R5_04_06 AT %I*: BOOL; //SPARE
	R5_04_07 AT %I*: BOOL; //SPARE

//***LCP4***BANK4 (Rack 6)****FORMATION****************************************************************
//EL3068 - AI1
	R6_01_00 		AT %I*: INT;
	R6_01_00_Status AT %I*: WORD;
	
	R6_01_01		AT %I*: INT;
	R6_01_01_Status AT %I*: WORD;
	
	R6_01_02 		AT %I*: INT;
	R6_01_02_Status AT %I*: WORD;
	
	R6_01_03 		AT %I*: INT;
	R6_01_03_Status AT %I*: WORD;
	
	R6_01_04 		AT %I*: INT;
	R6_01_04_Status AT %I*: WORD;
	
	R6_01_05 		AT %I*: INT;
	R6_01_05_Status AT %I*: WORD;
	
	R6_01_06 		AT %I*: INT;
	R6_01_06_Status AT %I*: WORD;
	
	R6_01_07 		AT %I*: INT;
	R6_01_07_Status AT %I*: WORD;
	
	//EL3068 - AI2
	R6_02_00 		AT %I*: INT;
	R6_02_00_Status AT %I*: WORD;
	
	R6_02_01		AT %I*: INT;
	R6_02_01_Status AT %I*: WORD;
	
	R6_02_02 		AT %I*: INT;
	R6_02_02_Status AT %I*: WORD;
	
	R6_02_03 		AT %I*: INT;
	R6_02_03_Status AT %I*: WORD;
	
	R6_02_04 		AT %I*: INT; 
	R6_02_04_Status AT %I*: WORD;
	
	R6_02_05 		AT %I*: INT; //SPARE
	R6_02_05_Status AT %I*: WORD;
	
	R6_02_06 		AT %I*: INT; //SPARE
	R6_02_06_Status AT %I*: WORD;
	
	R6_02_07 		AT %I*: INT; //SPARE
	R6_02_07_Status AT %I*: WORD;

//EL1008 - DI1
	R6_03_00 AT %I*: BOOL;
	R6_03_01 AT %I*: BOOL;
	R6_03_02 AT %I*: BOOL;
	R6_03_03 AT %I*: BOOL;
	R6_03_04 AT %I*: BOOL;
	R6_03_05 AT %I*: BOOL;
	R6_03_06 AT %I*: BOOL;
	R6_03_07 AT %I*: BOOL;
//EL1008 - DI2	
	R6_04_00 AT %I*: BOOL;
	R6_04_01 AT %I*: BOOL;
	R6_04_02 AT %I*: BOOL;
	R6_04_03 AT %I*: BOOL;
	R6_04_04 AT %I*: BOOL;
	R6_04_05 AT %I*: BOOL; 
	R6_04_06 AT %I*: BOOL; 
	R6_04_07 AT %I*: BOOL; 
//EL1008 - DI3	
	R6_05_00 AT %I*: BOOL;
	R6_05_01 AT %I*: BOOL;
	R6_05_02 AT %I*: BOOL;
	R6_05_03 AT %I*: BOOL;
	R6_05_04 AT %I*: BOOL; //spare
	R6_05_05 AT %I*: BOOL; //spare
	R6_05_06 AT %I*: BOOL; //spare
	R6_05_07 AT %I*: BOOL; //spare
//EL1008 - DI4	
	R6_06_00 AT %I*: BOOL;
	R6_06_01 AT %I*: BOOL;
	R6_06_02 AT %I*: BOOL;
	R6_06_03 AT %I*: BOOL;
	R6_06_04 AT %I*: BOOL; 
	R6_06_05 AT %I*: BOOL; 
	R6_06_06 AT %I*: BOOL; 
	R6_06_07 AT %I*: BOOL; 
//EL1008 - DI5	
	R6_07_00 AT %I*: BOOL;
	R6_07_01 AT %I*: BOOL;
	R6_07_02 AT %I*: BOOL;
	R6_07_03 AT %I*: BOOL; //spare
	R6_07_04 AT %I*: BOOL; //spare
	R6_07_05 AT %I*: BOOL; //spare
	R6_07_06 AT %I*: BOOL; //spare
	R6_07_07 AT %I*: BOOL; //spare

END_VAR

// ---- GVLs/InstrumentReading.TcGVL
{attribute 'qualified_only'}
VAR_GLOBAL
	//LCP 1 (Bank1 ) Instrument reading
	R2_03 : ST_InstrumentReading;
	//R2_02 : ARRAY [0..7] OF ST_InstrumentReading; // in case we need another card for R2
	R3_04 : ST_InstrumentReading;
	
END_VAR

// ---- GVLs/MCP_IO.TcGVL
{attribute 'qualified_only'}
VAR_GLOBAL
	MasterStopPB_Pressed		: BOOL;
	CageEstopCircuitOK			: BOOL;
	RemoteModeSelected			: BOOL;
	PSU1_DCOK					: BOOL;
	MachineGNDrlyOpen			: BOOL;
	//CloseAllChargeRlyCommand	: BOOL; only for slim
	//OpenAllDumpRelayCommand		: BOOL; only for slim
	//Charger 					: ARRAY [1..8] OF ST_Charger_Base;
	GLS3_Load					: ST_ChargeTime;
	GLS1_hvON					: BOOL;
	GLS2_hvON					: BOOL;
	GLS3_hvON					: BOOL;
	LiftMachineGND				: BOOL;
	//AllChargeRelaysClose		: BOOL; only for slim
	//AllDumpRelaysOpen			: BOOL; only for slim
	GLS1_voltageSP				: DINT;
	GLS1_voltageSP_norm			: REAL;
	GLS1_voltageSP_raw			: INT;
	
	GLS2_voltageSP				: DINT;
	GLS2_voltageSP_norm			: REAL;
	GLS2_voltageSP_raw			: INT;
	
	GLS3_voltageSP				: DINT;
	GLS3_voltageSP_norm			: REAL;
	GLS3_voltageSP_raw			: INT;

END_VAR

VAR_GLOBAL PERSISTENT
	Charger 					: ARRAY [1..8] OF ST_Charger_Base;
END_VAR

// ---- GVLs/Output.TcGVL
{attribute 'qualified_only'}
VAR_GLOBAL
	//***MCP Rack 2**************************************************
	//EL2008 - DQ1
	R2_01_00 AT %Q*: BOOL;
	R2_01_01 AT %Q*: BOOL;
	R2_01_02 AT %Q*: BOOL;
	R2_01_03 AT %Q*: BOOL;
	R2_01_04 AT %Q*: BOOL;
	R2_01_05 AT %Q*: BOOL;
	R2_01_06 AT %Q*: BOOL;
	R2_01_07 AT %Q*: BOOL;
	
	//EL2008 - DQ2
	R2_02_00 AT %Q*: BOOL;
	R2_02_01 AT %Q*: BOOL;
	R2_02_02 AT %Q*: BOOL;
	R2_02_03 AT %Q*: BOOL;
	R2_02_04 AT %Q*: BOOL;
	R2_02_05 AT %Q*: BOOL;
	R2_02_06 AT %Q*: BOOL;
	R2_02_07 AT %Q*: BOOL; 
	
	//EL4008 - AQ1
	R2_05_00 AT %Q*: INT;	//Charger 1 - Voltage Setpoint
	//R2_05_00_Status AT %Q*: WORD; //need to double check
	R2_05_01 AT %Q*: INT;	//Charger 2 - Voltage Setpoint
	//R2_05_01_Status AT %Q*: WORD;
	R2_05_02 AT %Q*: INT;	//Charger 3 - Voltage Setpoint
	//R2_05_02_Status AT %Q*: WORD;
	R2_05_03 AT %Q*: INT;	//Charger 4 - Voltage Setpoint
	//R2_05_03_Status AT %Q*: WORD;
	R2_05_04 AT %Q*: INT;	//Charger 5 - Voltage Setpoint
	//R2_05_04_Status AT %Q*: WORD;
	R2_05_05 AT %Q*: INT;	//Charger 6 - Voltage Setpoint
	//R2_05_05_Status AT %Q*: WORD;
	R2_05_06 AT %Q*: INT;	//Charger 7 - Voltage Setpoint
	//R2_05_06_Status AT %Q*: WORD;
	R2_05_07 AT %Q*: INT;	//Charger 8 - Voltage Setpoint
	//R2_05_07_Status AT %Q*: WORD;

	//EL2008 - DQ3
	R2_06_00 AT %Q*: BOOL;
	R2_06_01 AT %Q*: BOOL;
	R2_06_02 AT %Q*: BOOL;
	R2_06_03 AT %Q*: BOOL;  //Lift Machine Ground
	R2_06_04 AT %Q*: BOOL;  //spare
	R2_06_05 AT %Q*: BOOL;  //spare
	R2_06_06 AT %Q*: BOOL;  //spare
	R2_06_07 AT %Q*: BOOL;  //spare 

	//EL4008 - AQ2
	R2_07_00 AT %Q*: INT;	//GLS 1 - Voltage Setpoint
	//R2_07_00_Status AT %Q*: WORD; //need to double check
	R2_07_01 AT %Q*: INT;	//GLS 2 - Voltage Setpoint
	//R2_07_01_Status AT %Q*: WORD;
	R2_07_02 AT %Q*: INT;	//GLS 3 - Voltage Setpoint
	//R2_07_02_Status AT %Q*: WORD;
	R2_07_03 AT %Q*: INT;	//spare
	//R2_07_03_Status AT %Q*: WORD;
	R2_07_04 AT %Q*: INT;	//spare
	//R2_07_04_Status AT %Q*: WORD;
	R2_07_05 AT %Q*: INT;	//spare
	//R2_07_05_Status AT %Q*: WORD;
	R2_07_06 AT %Q*: INT;	//spare
	//R2_07_06_Status AT %Q*: WORD;
	R2_07_07 AT %Q*: INT;	//spare
	//R2_07_07_Status AT %Q*: WORD;
	
	//***LCP1***BANK1 (Rack 3)********************************************************************
	//EL2008 - DQ1
	R3_05_00 AT %Q*: BOOL;
	R3_05_01 AT %Q*: BOOL;
	R3_05_02 AT %Q*: BOOL;
	R3_05_03 AT %Q*: BOOL;
	R3_05_04 AT %Q*: BOOL;
	R3_05_05 AT %Q*: BOOL;
	R3_05_06 AT %Q*: BOOL;
	R3_05_07 AT %Q*: BOOL; 
	
	//EL2008 - DQ2
	R3_06_00 AT %Q*: BOOL; //BANK 1 SYSTEM READY TO CHARGE
	R3_06_01 AT %Q*: BOOL; //spare
	R3_06_02 AT %Q*: BOOL; //spare
	R3_06_03 AT %Q*: BOOL; //spare
	R3_06_04 AT %Q*: BOOL; //spare
	R3_06_05 AT %Q*: BOOL; //spare
	R3_06_06 AT %Q*: BOOL; //spare
	R3_06_07 AT %Q*: BOOL; //spare

	//***LCP2***BANK2 (Rack 4)********************************************************************
	//EL2008 - DQ1
	R4_05_00 AT %Q*: BOOL;
	R4_05_01 AT %Q*: BOOL;
	R4_05_02 AT %Q*: BOOL;
	R4_05_03 AT %Q*: BOOL;
	R4_05_04 AT %Q*: BOOL;
	R4_05_05 AT %Q*: BOOL;
	R4_05_06 AT %Q*: BOOL;
	R4_05_07 AT %Q*: BOOL; 
	
	//EL2008 - DQ2
	R4_06_00 AT %Q*: BOOL; //BANK 2 SYSTEM READY TO CHARGE
	R4_06_01 AT %Q*: BOOL; //spare
	R4_06_02 AT %Q*: BOOL; //spare
	R4_06_03 AT %Q*: BOOL; //spare
	R4_06_04 AT %Q*: BOOL; //spare
	R4_06_05 AT %Q*: BOOL; //spare
	R4_06_06 AT %Q*: BOOL; //spare
	R4_06_07 AT %Q*: BOOL; //spare
	
	//***LCP3***BANK3 (Rack 5)********************************************************************
	//EL2008 - DQ1
	R5_05_00 AT %Q*: BOOL;
	R5_05_01 AT %Q*: BOOL;
	R5_05_02 AT %Q*: BOOL;
	R5_05_03 AT %Q*: BOOL;
	R5_05_04 AT %Q*: BOOL;
	R5_05_05 AT %Q*: BOOL;
	R5_05_06 AT %Q*: BOOL;
	R5_05_07 AT %Q*: BOOL; 
	
	//EL2008 - DQ2
	R5_06_00 AT %Q*: BOOL; //BANK 3 SYSTEM READY TO CHARGE
	R5_06_01 AT %Q*: BOOL; //spare
	R5_06_02 AT %Q*: BOOL; //spare
	R5_06_03 AT %Q*: BOOL; //spare
	R5_06_04 AT %Q*: BOOL; //spare
	R5_06_05 AT %Q*: BOOL; //spare
	R5_06_06 AT %Q*: BOOL; //spare
	R5_06_07 AT %Q*: BOOL; //spare

	//***LCP4***BANK4 (Rack 6)*******Formation*************************************************************
	//EL2008 - DQ1
	R6_06_00 AT %Q*: BOOL;
	R6_06_01 AT %Q*: BOOL;
	R6_06_02 AT %Q*: BOOL;
	R6_06_03 AT %Q*: BOOL;
	R6_06_04 AT %Q*: BOOL;
	R6_06_05 AT %Q*: BOOL;
	R6_06_06 AT %Q*: BOOL;
	R6_06_07 AT %Q*: BOOL; 
	
	//EL2008 - DQ2
	R6_07_00 AT %Q*: BOOL; 
	R6_07_01 AT %Q*: BOOL; 
	R6_07_02 AT %Q*: BOOL; 
	R6_07_03 AT %Q*: BOOL; //spare
	R6_07_04 AT %Q*: BOOL; //spare
	R6_07_05 AT %Q*: BOOL; //spare
	R6_07_06 AT %Q*: BOOL; //spare
	R6_07_07 AT %Q*: BOOL; //spare
	
END_VAR

// ---- GVLs/Permissives_DB.TcGVL
{attribute 'qualified_only'}
VAR_GLOBAL
	AllShortContactEngaged	: BOOL;
	AllDumpRelaysOpen		: BOOL;
	AllChargeRelaysClosed	: BOOL;
	AllSystemsReadytoCharge	: BOOL;
	NoShortingUnknowns		: BOOL;
	AllChargerInhibited		: BOOL;
	AllChargerHVisON		: BOOL;
	AllSectCapsDischarged	: BOOL;
	AllSectCapsFullyCharged : BOOL;
	NoInterlockPressureLoss : BOOL;
	SafetyOK				: BOOL;
	AllChargerEOC			: BOOL;
	
	AllSection1ChargeRlyClose : BOOL;
	AllSection2ChargeRlyClose : BOOL;
	AllSection3ChargeRlyClose : BOOL;
	AllSection4ChargeRlyClose : BOOL;
	
	AllSection1DumpRlyOpen : BOOL;
	AllSection2DumpRlyOpen : BOOL;
	AllSection3DumpRlyOpen : BOOL;
	AllSection4DumpRlyOpen : BOOL;
	
	AllPeakChargeRlyClose	: BOOL;
	AllSustChargeRlyClose	: BOOL;
	AllFormChargeRlyClose	: BOOL;
	
	AllPeakDumpRlyOpen		: BOOL;
	AllSustDumpRlyOpen		: BOOL;
	AllFormDumpRlyOpen		: BOOL;
	
	AllPeakChargerHVisON	: BOOL;
	AllSustChargerHVisOn	: BOOL;
	AllFormChargerHVisOn	: BOOL;
	
	AllPeakChargerInhibited : BOOL;
	AllSustChargerInhibited	: BOOL;
	AllFormChargerInhibited : BOOL;
	
END_VAR

// ---- GVLs/Trips_DB.TcGVL
{attribute 'qualified_only'}
VAR_GLOBAL
	Section 					: ARRAY[1..4] OF ST_Trip_Base;
	Charger						: ARRAY[1..8] OF ST_Charger_Base;
	MasterStopPBPressed			: BOOL;
	CageEStopCircuitBroken		: BOOL;
	LocalModeSelected			: BOOL;
	MCPLossDCpower				: BOOL;
	MCPsystemTripped			: BOOL;
	
	AnyEstopPressed 			: BOOL;
	AllDCpsuOK					: BOOL;
	AnyChargerOverTemp			: BOOL;
	AnyChargerLoadFault			: BOOL;
	AnyChargerInterlockOpen		: BOOL;
	AnyChargerFaulted			: BOOL; // same as summary fault
	AnySystemTripped			: BOOL; //LCP 1-4
	MachineGNDrlyFailed			: BOOL;
	//SystemTripped 				: BOOL;
	//InstrumentationFaulted		: BOOL;
	AnyChargeRlyFail			: BOOL;
	AnyDumpRlyFail				: BOOL;
	//AnyACInterlockFail			: BOOL;
	AnyLossInhibitSignal		: BOOL;
	AnyLossHVONsignal			: BOOL;
	
	ChargingTimerRunout         : BOOL;
	ChargedTimerRunout			: BOOL;
	DumpTimerRunout				: BOOL;
	//SystemTimeOut				: BOOL;
	NoFaultDetected				: BOOL;
	ClearAllFaults				: BOOL;
END_VAR

// ---- POUs/MAIN.TcPOU
PROGRAM MAIN
VAR
END_VAR

Alias();
//Heartbeat_1();
Permissives();
Trips();
Alarms();
Sequence();
Communication();
Analogconversion();
HMI();
ChargeTime();

END_PROGRAM

// ---- POUs/Alias.TcPOU
PROGRAM Alias
VAR
END_VAR

//R1 & R2 : MCP**  
	//DI
	MCP_IO.MasterStopPB_Pressed					:= NOT Input.R1_01_00;  //NC - Master stop PB not pressed - black pb on mcp
	MCP_IO.CageEstopCircuitOK					:= Input.R1_01_01;  //case Estop circuit okay (Rly1 (120vac)
	MCP_IO.RemoteModeSelected					:= Input.R1_01_02; // 0 = manual, 1=auto
	MCP_IO.PSU1_DCOK							:= Input.R1_01_03; //psu1 dc ok
	MCP_IO.MachineGNDrlyOpen					:= Input.R1_01_04; // machine ground lifted (opto board)	
	//MCP_IO.CloseAllChargeRlyCommand				:= Input.R1_01_05; // command from screen room (opto) - Slim only
	//MCP_IO.OpenAllDumpRelayCommand				:= Input.R1_01_06; // command from screen room (opto) - slim only
	
	MCP_IO.Charger[1].inhibited					:= NOT Input.R1_02_00; //TDK802 1
	MCP_IO.Charger[1].EndOfCharge				:= NOT Input.R1_02_01; //TDK802 1
	MCP_IO.Charger[1].HV_isON					:= NOT Input.R1_02_02; //TDK802 1
	MCP_IO.Charger[1].OverTemp					:= NOT Input.R1_02_03; //TDK802 1
	MCP_IO.Charger[1].InterlockOpen				:= NOT Input.R1_02_04; //TDK802 1
	MCP_IO.Charger[1].LoadFaulted				:= NOT Input.R1_02_05; //TDK802 1
	MCP_IO.Charger[1].SummaryFaulted			:= NOT Input.R1_02_06; //TDK802 1
	
	MCP_IO.Charger[2].inhibited					:= NOT Input.R1_03_00; //TDK802 2
	MCP_IO.Charger[2].EndOfCharge				:= NOT Input.R1_03_01; 
	MCP_IO.Charger[2].HV_isON					:= NOT Input.R1_03_02; 
	MCP_IO.Charger[2].OverTemp					:= NOT Input.R1_03_03; 
	MCP_IO.Charger[2].InterlockOpen				:= NOT Input.R1_03_04; 
	MCP_IO.Charger[2].LoadFaulted				:= NOT Input.R1_03_05; 
	MCP_IO.Charger[2].SummaryFaulted			:= NOT Input.R1_03_06; 
	
	MCP_IO.Charger[3].inhibited					:= NOT Input.R1_04_00; //TDK802 3
	MCP_IO.Charger[3].EndOfCharge				:= NOT Input.R1_04_01; 
	MCP_IO.Charger[3].HV_isON					:= NOT Input.R1_04_02; 
	MCP_IO.Charger[3].OverTemp					:= NOT Input.R1_04_03; 
	MCP_IO.Charger[3].InterlockOpen				:= NOT Input.R1_04_04; 
	MCP_IO.Charger[3].LoadFaulted				:= NOT Input.R1_04_05; 
	MCP_IO.Charger[3].SummaryFaulted			:= NOT Input.R1_04_06; 
	
	MCP_IO.Charger[4].inhibited					:= NOT Input.R1_05_00; //TDK802 4
	MCP_IO.Charger[4].EndOfCharge				:= NOT Input.R1_05_01; 
	MCP_IO.Charger[4].HV_isON					:= NOT Input.R1_05_02; 
	MCP_IO.Charger[4].OverTemp					:= NOT Input.R1_05_03; 
	MCP_IO.Charger[4].InterlockOpen				:= NOT Input.R1_05_04; 
	MCP_IO.Charger[4].LoadFaulted				:= NOT Input.R1_05_05; 
	MCP_IO.Charger[4].SummaryFaulted			:= NOT Input.R1_05_06; 

	MCP_IO.Charger[5].inhibited					:= NOT Input.R1_06_00; //TDK802 5
	MCP_IO.Charger[5].EndOfCharge				:= NOT Input.R1_06_01; 
	MCP_IO.Charger[5].HV_isON					:= NOT Input.R1_06_02; 
	MCP_IO.Charger[5].OverTemp					:= NOT Input.R1_06_03; 
	MCP_IO.Charger[5].InterlockOpen				:= NOT Input.R1_06_04; 
	MCP_IO.Charger[5].LoadFaulted				:= NOT Input.R1_06_05; 
	MCP_IO.Charger[5].SummaryFaulted			:= NOT Input.R1_06_06; 

	MCP_IO.Charger[6].inhibited					:= NOT Input.R1_07_00; //TDK802 6
	MCP_IO.Charger[6].EndOfCharge				:= NOT Input.R1_07_01; 
	MCP_IO.Charger[6].HV_isON					:= NOT Input.R1_07_02; 
	MCP_IO.Charger[6].OverTemp					:= NOT Input.R1_07_03; 
	MCP_IO.Charger[6].InterlockOpen				:= NOT Input.R1_07_04; 
	MCP_IO.Charger[6].LoadFaulted				:= NOT Input.R1_07_05; 
	MCP_IO.Charger[6].SummaryFaulted			:= NOT Input.R1_07_06; 

	MCP_IO.Charger[7].inhibited					:= NOT Input.R1_08_00; //TDK802 7
	MCP_IO.Charger[7].EndOfCharge				:= NOT Input.R1_08_01; 
	MCP_IO.Charger[7].HV_isON					:= NOT Input.R1_08_02; 
	MCP_IO.Charger[7].OverTemp					:= NOT Input.R1_08_03; 
	MCP_IO.Charger[7].InterlockOpen				:= NOT Input.R1_08_04; 
	MCP_IO.Charger[7].LoadFaulted				:= NOT Input.R1_08_05; 
	MCP_IO.Charger[7].SummaryFaulted			:= NOT Input.R1_08_06; 

	MCP_IO.Charger[8].inhibited					:= NOT Input.R1_09_00; //TDK802 8
	MCP_IO.Charger[8].EndOfCharge				:= NOT Input.R1_09_01; 
	MCP_IO.Charger[8].HV_isON					:= NOT Input.R1_09_02; 
	MCP_IO.Charger[8].OverTemp					:= NOT Input.R1_09_03; 
	MCP_IO.Charger[8].InterlockOpen				:= NOT Input.R1_09_04; 
	MCP_IO.Charger[8].LoadFaulted				:= NOT Input.R1_09_05; 
	MCP_IO.Charger[8].SummaryFaulted			:= NOT Input.R1_09_06; 
	
	//DQ
	Output.R2_01_00	:= MCP_IO.Charger[1].inhibit;
	Output.R2_01_01	:= MCP_IO.Charger[1].HV_ON;
	Output.R2_01_02	:= MCP_IO.Charger[2].inhibit;
	Output.R2_01_03	:= MCP_IO.Charger[2].HV_ON;
	Output.R2_01_04	:= MCP_IO.Charger[3].inhibit;
	Output.R2_01_05	:= MCP_IO.Charger[3].HV_ON;
	Output.R2_01_06	:= MCP_IO.Charger[4].inhibit;
	Output.R2_01_07	:= MCP_IO.Charger[4].HV_ON;
	
	Output.R2_02_00	:= MCP_IO.Charger[5].inhibit;
	Output.R2_02_01	:= MCP_IO.Charger[5].HV_ON;
	Output.R2_02_02	:= MCP_IO.Charger[6].inhibit;
	Output.R2_02_03	:= MCP_IO.Charger[6].HV_ON;
	Output.R2_02_04	:= MCP_IO.Charger[7].inhibit;
	Output.R2_02_05	:= MCP_IO.Charger[7].HV_ON;
	Output.R2_02_06	:= MCP_IO.Charger[8].inhibit;
	Output.R2_02_07	:= MCP_IO.Charger[8].HV_ON;
	
	//AI
	MCP_IO.Charger[1].voltageFeedback_raw		:= Input.R2_03_00;
	MCP_IO.Charger[1].currentFeedback_raw		:= Input.R2_03_01;
	MCP_IO.Charger[2].voltageFeedback_raw		:= Input.R2_03_02;
	MCP_IO.Charger[2].currentFeedback_raw		:= Input.R2_03_03;
	MCP_IO.Charger[3].voltageFeedback_raw		:= Input.R2_03_04;
	MCP_IO.Charger[3].currentFeedback_raw		:= Input.R2_03_05;
	MCP_IO.Charger[4].voltageFeedback_raw		:= Input.R2_03_06;
	MCP_IO.Charger[4].currentFeedback_raw		:= Input.R2_03_07;
	
	MCP_IO.Charger[5].voltageFeedback_raw		:= Input.R2_04_00;
	MCP_IO.Charger[5].currentFeedback_raw		:= Input.R2_04_01;
	MCP_IO.Charger[6].voltageFeedback_raw		:= Input.R2_04_02;
	MCP_IO.Charger[6].currentFeedback_raw		:= Input.R2_04_03;
	MCP_IO.Charger[7].voltageFeedback_raw		:= Input.R2_04_04;
	MCP_IO.Charger[7].currentFeedback_raw		:= Input.R2_04_05;
	MCP_IO.Charger[8].voltageFeedback_raw		:= Input.R2_04_06;
	MCP_IO.Charger[8].currentFeedback_raw		:= Input.R2_04_07;
	
	//AQ
	Output.R2_05_00	:= MCP_IO.Charger[1].voltageSP_raw;
	Output.R2_05_01	:= MCP_IO.Charger[2].voltageSP_raw;
	Output.R2_05_02	:= MCP_IO.Charger[3].voltageSP_raw;
	Output.R2_05_03	:= MCP_IO.Charger[4].voltageSP_raw;	
	Output.R2_05_04	:= MCP_IO.Charger[5].voltageSP_raw;
	Output.R2_05_05	:= MCP_IO.Charger[6].voltageSP_raw;
	Output.R2_05_06	:= MCP_IO.Charger[7].voltageSP_raw;
	Output.R2_05_07	:= MCP_IO.Charger[8].voltageSP_raw;	
	
	Output.R2_06_00	:= MCP_IO.GLS1_hvON;
	Output.R2_06_01	:= MCP_IO.GLS2_hvON;
	Output.R2_06_02	:= MCP_IO.GLS3_hvON;
	Output.R2_06_03	:= MCP_IO.LiftMachineGND;
	//Output.R2_06_04	:= MCP_IO.AllChargeRelaysClose; //only for slim
	//Output.R2_06_05	:= MCP_IO.AllDumpRelaysOpen;  // only for slim				
	
	Output.R2_07_00	:= MCP_IO.GLS1_voltageSP_raw; //Form Trigger
	Output.R2_07_01	:= MCP_IO.GLS2_voltageSP_raw;  //Preform trigger
	Output.R2_07_02	:= MCP_IO.GLS3_voltageSP_raw; //preform cap charger

//R3 : Bank 1 (LCP1)***********************************************
	//EL3068 - AI
	LCP.Section[1].Peak.cap[1].voltageFeedback_raw := Input.R3_01_00;
	LCP.Section[1].Peak.cap[2].voltageFeedback_raw := Input.R3_01_01;
	LCP.Section[1].Peak.cap[3].voltageFeedback_raw := Input.R3_01_02;
	LCP.Section[1].Peak.cap[4].voltageFeedback_raw := Input.R3_01_03;
	LCP.Section[1].Peak.cap[5].voltageFeedback_raw := Input.R3_01_04;
	LCP.Section[1].Peak.cap[6].voltageFeedback_raw := Input.R3_01_05;
	LCP.Section[1].Peak.cap[7].voltageFeedback_raw := Input.R3_01_06;
	LCP.Section[1].Peak.cap[8].voltageFeedback_raw := Input.R3_01_07;
	LCP.Section[1].Peak.cap[9].voltageFeedback_raw := Input.R3_02_00;
	LCP.Section[1].Peak.cap[10].voltageFeedback_raw := Input.R3_02_01;
	
	LCP.Section[1].Sust.cap[1].voltageFeedback_raw := Input.R3_02_02;
	LCP.Section[1].Sust.cap[2].voltageFeedback_raw := Input.R3_02_03;
	
	//DI
	LCP.Section[1].Peak.ChargeRelay1_close 	:= Input.R3_03_00; //RLY 1A
	LCP.Section[1].Peak.ChargeRelay2_close 	:= Input.R3_03_01; //RLY 2A
	LCP.Section[1].Peak.DumpRelay1_close 	:= Input.R3_03_02; //RLY 3A
	LCP.Section[1].Peak.DumpRelay2_close	:= Input.R3_03_03; //RLY 4A
	LCP.Section[1].Sust.ChargeRelay1_close	:= Input.R3_03_04; //RLY 5A
	LCP.Section[1].Sust.ChargeRelay2_close	:= Input.R3_03_05; //RLY 6A
	LCP.Section[1].Sust.DumpRelay1_close	:= Input.R3_03_06; //RLY 7A
	LCP.Section[1].Sust.DumpRelay2_close	:= Input.R3_03_07; //RLY 8A
	
	LCP.Section[1].Peak.ShortContact1_close 	:= Input.R3_04_00; //psw1
	LCP.Section[1].Peak.UnshortContact1_close 	:= Input.R3_04_01; //psw2
	LCP.Section[1].Peak.ShortContact2_close 	:= Input.R3_04_02; //psw3
	LCP.Section[1].Peak.UnshortContact2_close 	:= Input.R3_04_03; //psw4
	LCP.Section[1].LossPneumaticPressure 		:= Input.R3_04_04; //psw5
	LCP.Section[1].PSU1_DCOK					:= Input.R3_04_05; //psu1 contact

	//DQ
	Output.R3_05_00 := LCP.Section[1].Peak.CloseChargeRelay1; //RLY1
	Output.R3_05_01 := LCP.Section[1].Peak.CloseChargeRelay2; //RLY2
	Output.R3_05_02 := LCP.Section[1].Peak.OpenDumpRelay1; //RLY3
	Output.R3_05_03 := LCP.Section[1].Peak.OpenDumpRelay2; //RLY4
	Output.R3_05_04 := LCP.Section[1].Sust.CloseChargeRelay1; //RLY5
	Output.R3_05_05 := LCP.Section[1].Sust.CloseChargeRelay2; //RLY6
	Output.R3_05_06 := LCP.Section[1].Sust.OpenDumpRelay1; //RLY7
	Output.R3_05_07 := LCP.Section[1].Sust.OpenDumpRelay2; //RLY8
	Output.R3_06_00 := LCP.Section[1].SystemReadyToCharge; //LED1

//R4 : Bank 2 (LCP2)***********************************************
	//EL3068 - AI
	LCP.Section[2].Peak.cap[1].voltageFeedback_raw := Input.R4_01_00;
	LCP.Section[2].Peak.cap[2].voltageFeedback_raw := Input.R4_01_01;
	LCP.Section[2].Peak.cap[3].voltageFeedback_raw := Input.R4_01_02;
	LCP.Section[2].Peak.cap[4].voltageFeedback_raw := Input.R4_01_03;
	LCP.Section[2].Peak.cap[5].voltageFeedback_raw := Input.R4_01_04;
	LCP.Section[2].Peak.cap[6].voltageFeedback_raw := Input.R4_01_05;
	LCP.Section[2].Peak.cap[7].voltageFeedback_raw := Input.R4_01_06;
	LCP.Section[2].Peak.cap[8].voltageFeedback_raw := Input.R4_01_07;
	LCP.Section[2].Peak.cap[9].voltageFeedback_raw := Input.R4_02_00;
	LCP.Section[2].Peak.cap[10].voltageFeedback_raw := Input.R4_02_01;
	
	LCP.Section[2].Sust.cap[1].voltageFeedback_raw := Input.R4_02_02;
	LCP.Section[2].Sust.cap[2].voltageFeedback_raw := Input.R4_02_03;
	
	//DI
	LCP.Section[2].Peak.ChargeRelay1_close 	:= Input.R4_03_00; //RLY 1A
	LCP.Section[2].Peak.ChargeRelay2_close 	:= Input.R4_03_01; //RLY 2A
	LCP.Section[2].Peak.DumpRelay1_close 	:= Input.R4_03_02; //RLY 3A
	LCP.Section[2].Peak.DumpRelay2_close	:= Input.R4_03_03; //RLY 4A
	LCP.Section[2].Sust.ChargeRelay1_close	:= Input.R4_03_04; //RLY 5A
	LCP.Section[2].Sust.ChargeRelay2_close	:= Input.R4_03_05; //RLY 6A
	LCP.Section[2].Sust.DumpRelay1_close	:= Input.R4_03_06; //RLY 7A
	LCP.Section[2].Sust.DumpRelay2_close	:= Input.R4_03_07; //RLY 8A
	
	LCP.Section[2].Peak.ShortContact1_close 	:= Input.R4_04_00; //psw1
	LCP.Section[2].Peak.UnshortContact1_close 	:= Input.R4_04_01; //psw2
	LCP.Section[2].Peak.ShortContact2_close 	:= Input.R4_04_02; //psw3
	LCP.Section[2].Peak.UnshortContact2_close 	:= Input.R4_04_03; //psw4
	LCP.Section[2].LossPneumaticPressure 		:= Input.R4_04_04; //psw5
	LCP.Section[2].PSU1_DCOK					:= Input.R4_04_05; //psu1 contact

	//DQ
	Output.R4_05_00 := LCP.Section[2].Peak.CloseChargeRelay1; //RLY1
	Output.R4_05_01 := LCP.Section[2].Peak.CloseChargeRelay2; //RLY2
	Output.R4_05_02 := LCP.Section[2].Peak.OpenDumpRelay1; //RLY3
	Output.R4_05_03 := LCP.Section[2].Peak.OpenDumpRelay2; //RLY4
	Output.R4_05_04 := LCP.Section[2].Sust.CloseChargeRelay1; //RLY5
	Output.R4_05_05 := LCP.Section[2].Sust.CloseChargeRelay2; //RLY6
	Output.R4_05_06 := LCP.Section[2].Sust.OpenDumpRelay1; //RLY7
	Output.R4_05_07 := LCP.Section[2].Sust.OpenDumpRelay2; //RLY8
	Output.R4_06_00 := LCP.Section[2].SystemReadyToCharge; //LED1

//R5 : Bank 3 (LCP3)***********************************************
	//EL3068 - AI
	LCP.Section[3].Peak.cap[1].voltageFeedback_raw := Input.R5_01_00;
	LCP.Section[3].Peak.cap[2].voltageFeedback_raw := Input.R5_01_01;
	LCP.Section[3].Peak.cap[3].voltageFeedback_raw := Input.R5_01_02;
	LCP.Section[3].Peak.cap[4].voltageFeedback_raw := Input.R5_01_03;
	LCP.Section[3].Peak.cap[5].voltageFeedback_raw := Input.R5_01_04;
	LCP.Section[3].Peak.cap[6].voltageFeedback_raw := Input.R5_01_05;
	LCP.Section[3].Peak.cap[7].voltageFeedback_raw := Input.R5_01_06;
	LCP.Section[3].Peak.cap[8].voltageFeedback_raw := Input.R5_01_07;
	LCP.Section[3].Peak.cap[9].voltageFeedback_raw := Input.R5_02_00;
	LCP.Section[3].Peak.cap[10].voltageFeedback_raw := Input.R5_02_01;
	
	LCP.Section[3].Sust.cap[1].voltageFeedback_raw := Input.R5_02_02;
	LCP.Section[3].Sust.cap[2].voltageFeedback_raw := Input.R5_02_03;
	
	//DI
	LCP.Section[3].Peak.ChargeRelay1_close 	:= Input.R5_03_00; //RLY 1A
	LCP.Section[3].Peak.ChargeRelay2_close 	:= Input.R5_03_01; //RLY 2A
	LCP.Section[3].Peak.DumpRelay1_close 	:= Input.R5_03_02; //RLY 3A
	LCP.Section[3].Peak.DumpRelay2_close	:= Input.R5_03_03; //RLY 4A
	LCP.Section[3].Sust.ChargeRelay1_close	:= Input.R5_03_04; //RLY 5A
	LCP.Section[3].Sust.ChargeRelay2_close	:= Input.R5_03_05; //RLY 6A
	LCP.Section[3].Sust.DumpRelay1_close	:= Input.R5_03_06; //RLY 7A
	LCP.Section[3].Sust.DumpRelay2_close	:= Input.R5_03_07; //RLY 8A
	
	LCP.Section[3].Peak.ShortContact1_close 	:= Input.R5_04_00; //psw1
	LCP.Section[3].Peak.UnshortContact1_close 	:= Input.R5_04_01; //psw2
	LCP.Section[3].Peak.ShortContact2_close 	:= Input.R5_04_02; //psw3
	LCP.Section[3].Peak.UnshortContact2_close 	:= Input.R5_04_03; //psw4
	LCP.Section[3].LossPneumaticPressure 		:= Input.R5_04_04; //psw5
	LCP.Section[3].PSU1_DCOK					:= Input.R5_04_05; //psu1 contact

	//DQ
	Output.R5_05_00 := LCP.Section[3].Peak.CloseChargeRelay1; //RLY1
	Output.R5_05_01 := LCP.Section[3].Peak.CloseChargeRelay2; //RLY2
	Output.R5_05_02 := LCP.Section[3].Peak.OpenDumpRelay1; //RLY3
	Output.R5_05_03 := LCP.Section[3].Peak.OpenDumpRelay2; //RLY4
	Output.R5_05_04 := LCP.Section[3].Sust.CloseChargeRelay1; //RLY5
	Output.R5_05_05 := LCP.Section[3].Sust.CloseChargeRelay2; //RLY6
	Output.R5_05_06 := LCP.Section[3].Sust.OpenDumpRelay1; //RLY7
	Output.R5_05_07 := LCP.Section[3].Sust.OpenDumpRelay2; //RLY8
	Output.R5_06_00 := LCP.Section[3].SystemReadyToCharge; //LED1

//R6 : Bank 4 (LCP4)*****Formation******************************************
	//EL3068 - AI
	LCP.Section[4].Form.cap[1].voltageFeedback_raw := Input.R6_01_00;
	LCP.Section[4].Form.cap[2].voltageFeedback_raw := Input.R6_01_01;
	LCP.Section[4].Form.cap[3].voltageFeedback_raw := Input.R6_01_02;
	LCP.Section[4].Form.cap[4].voltageFeedback_raw := Input.R6_01_03;
	LCP.Section[4].Form.cap[5].voltageFeedback_raw := Input.R6_01_04;
	LCP.Section[4].Form.cap[6].voltageFeedback_raw := Input.R6_01_05;
	LCP.Section[4].Form.cap[7].voltageFeedback_raw := Input.R6_01_06;
	LCP.Section[4].Form.cap[8].voltageFeedback_raw := Input.R6_01_07;
	
	LCP.Section[4].Form.cap[9].voltageFeedback_raw	:= Input.R6_02_00;
	LCP.Section[4].Form.cap[10].voltageFeedback_raw := Input.R6_02_01;
	LCP.Section[4].Form.cap[11].voltageFeedback_raw := Input.R6_02_02;
	LCP.Section[4].Form.cap[12].voltageFeedback_raw := Input.R6_02_03;
	LCP.Section[4].FormTriggerVoltage_raw		 	:= Input.R6_02_04;
	LCP.Section[4].PreFormTriggerVoltage_raw	 	:= Input.R6_02_05;
	LCP.Section[4].PreFormCapVoltage_raw		 	:= Input.R6_02_06;
	
	
	//DI
	LCP.Section[4].Form.ChargeRelay1_close			:= Input.R6_03_00;	//RLY 1A
	LCP.Section[4].Form.ChargeRelay2_close			:= Input.R6_03_01;	//RLY 2A
	LCP.Section[4].Form.PreFormChargeRly_close		:= Input.R6_03_02;	//RLY 3A	
	LCP.Section[4].Form.FormTrigChargeRly_close		:= Input.R6_03_03;	//RLY 4A
	LCP.Section[4].Form.PreFormTrigChargeRly_close	:= Input.R6_03_04;	//RLY 5A
	LCP.Section[4].Form.DumpRelay1_close			:= Input.R6_03_05;	//RLY 6A
	LCP.Section[4].Form.DumpRelay2_close			:= Input.R6_03_06;	//RLY 7A
	LCP.Section[4].Form.PreFormDumpRly_close		:= Input.R6_03_07;	//RLY 8A
	LCP.Section[4].Form.FormTrigDumpRly1_close		:= Input.R6_04_00;	//RLY 9A
	LCP.Section[4].Form.PreFormTrigDumpRly1_close	:= Input.R6_04_01;	//RLY 10A
	
	LCP.Section[4].Form.ShortContact1_close		:= Input.R6_04_02;  //psw1
	LCP.Section[4].Form.UnshortContact1_close	:= Input.R6_04_03;  //psw2
	LCP.Section[4].Form.ShortContact2_close		:= Input.R6_04_04;  //psw3
	LCP.Section[4].Form.UnshortContact2_close	:= Input.R6_04_05;  //psw4
	LCP.Section[4].Form.FormTrigShortContact_close		:= Input.R6_04_06;  //psw5
	LCP.Section[4].Form.FormTrigUnshortContact_close	:= Input.R6_04_07;  //psw6
	LCP.Section[4].Form.PreFormTrigShortContact_close	:= Input.R6_05_00;  //psw7
	LCP.Section[4].Form.PreFormTrigUnShortContact_close	:= Input.R6_05_01;  //psw8
	LCP.Section[4].LossPneumaticPressure				:= Input.R6_05_02;  //psw9
	LCP.Section[4].PSU1_DCOK							:= Input.R6_05_03;  //psu1
	
	//DQ
	Output.R6_06_00 := LCP.Section[4].Form.CloseChargeRelay1; //rly1
	Output.R6_06_01 := LCP.Section[4].Form.CloseChargeRelay2; //rly2
	Output.R6_06_02 := LCP.Section[4].Form.ClosePreFormChargeRly; //rly3
	Output.R6_06_03 := LCP.Section[4].Form.CloseFormTrigChargeRly; //rly4
	Output.R6_06_04 := LCP.Section[4].Form.ClosePreFormTrigChargeRly; //rly5
	Output.R6_06_05 := LCP.Section[4].Form.OpenDumpRelay1; //rly6
	Output.R6_06_06 := LCP.Section[4].Form.OpenDumpRelay2; //rly7
	Output.R6_06_07 := LCP.Section[4].Form.OpenPreFormDumpRly; //rly8
	
	Output.R6_07_00 := LCP.Section[4].Form.OpenFormTrigDumpRly1; //rly9
	Output.R6_07_01 := LCP.Section[4].Form.OpenPreFormTrigDumpRly1; //rly10
	Output.R6_07_02 := LCP.Section[4].SystemReadyToCharge; //LED1
	
	//InstrumentReading.R2_01_CH00 := Input.R3_01_00;
	//InstrumentReading.R2_01_CH01 := Input.R3_01_01;
	(*
	R2_01_02 		AT %I*: INT;
	R2_01_02_Status AT %I*: WORD;
	
	R2_01_03 		AT %I*: INT;
	R2_01_03_Status AT %I*: WORD;
	
	R2_01_04 		AT %I*: INT;
	R2_01_04_Status AT %I*: WORD;
	
	R2_01_05 		AT %I*: INT;
	R2_01_05_Status AT %I*: WORD;
	
	R2_01_06 		AT %I*: INT;
	R2_01_06_Status AT %I*: WORD;
	
	R2_01_07 		AT %I*: INT;
	R2_01_07_Status AT %I*: WORD;
	*)

END_PROGRAM

// ---- POUs/Permissives.TcPOU
PROGRAM Permissives
VAR
	i : INT := 1;  //for section 1 - 3 
	j : INT := 1; //for charger 1-8
	k : INT := 1; //cap 1- 10
	m : INT := 1; //form cap 1-12
	n : INT := 1; //1-6
	p : INT := 7; //7-12
END_VAR

//Charger summary faults
//Trips_DB.AnySummaryFault = FALSE AND Trips_DB.AnyEstopPressed //add to no fault detected.

//section ready to charge
FOR i := 1 TO 3 BY 1 DO
	IF Trips_DB.NoFaultDetected = TRUE AND //MCP_IO.Charger[1-8].HVisOn AND
		Permissives_DB.AllChargeRelaysClosed = TRUE AND
		LCP.Section[i].Peak.ShortContact1Engaged = FALSE AND
		LCP.Section[i].Peak.ShortContact2Engaged = FALSE AND
		LCP.Section[i].Sust.ShortContact1Engaged = FALSE AND
		LCP.Section[i].Sust.ShortContact2Engaged = FALSE
	THEN
		LCP.Section[i].SystemReadyToCharge := TRUE;	
	ELSE
		LCP.Section[i].SystemReadyToCharge := FALSE;		
	END_IF;
END_FOR;

//Section 4
IF Trips_DB.NoFaultDetected = TRUE AND //MCP_IO.Charger[1-8].HVisOn AND
	Permissives_DB.AllChargeRelaysClosed = TRUE AND
	LCP.Section[4].Form.ShortContact1Engaged = FALSE AND
	LCP.Section[4].Form.ShortContact2Engaged = FALSE AND
	LCP.Section[4].Form.FormTrigShortContactEngaged = FALSE AND
	LCP.Section[4].Form.PreFormTrigShortContactEngaged = FALSE 
	THEN
		LCP.Section[4].SystemReadyToCharge := TRUE;
	ELSE
		LCP.Section[4].SystemReadyToCharge := FALSE;
END_IF;
	
IF LCP.Section[1].SystemReadyToCharge = TRUE AND 
	LCP.Section[2].SystemReadyToCharge = TRUE AND
	LCP.Section[3].SystemReadyToCharge = TRUE AND
	LCP.Section[4].SystemReadyToCharge = TRUE
	THEN
		Permissives_DB.AllSystemsReadytoCharge := TRUE;
		ELSE
			Permissives_DB.AllSystemsReadytoCharge := FALSE;
END_IF


// shorts and unshorts
//Peaking  -- short contacts are NO, so if close is false, it is and unshort is true, then it is not shorted 
FOR i := 1 TO 3 BY 1 DO
	IF LCP.Section[i].Peak.ShortContact1_close = TRUE AND LCP.Section[i].Peak.UnshortContact1_close = FALSE 
		THEN
			LCP.Section[i].Peak.ShortContact1Engaged := TRUE;
		ELSE
			LCP.Section[i].Peak.ShortContact1Engaged := FALSE;
	END_IF;
	
	IF LCP.Section[i].Peak.ShortContact2_close = TRUE AND LCP.Section[i].Peak.UnshortContact2_close = FALSE 
		THEN
			LCP.Section[i].Peak.ShortContact2Engaged := TRUE;
		ELSE
			LCP.Section[i].Peak.ShortContact2Engaged := FALSE;
	END_IF;
	
END_FOR;

//Sustain
FOR i := 1 TO 3 BY 1 DO
	IF LCP.Section[i].Sust.ShortContact1_close = TRUE AND LCP.Section[i].Sust.UnshortContact1_close = FALSE 
		THEN
			LCP.Section[i].Sust.ShortContact1Engaged := TRUE;
		ELSE
			LCP.Section[i].Sust.ShortContact1Engaged := FALSE;
	END_IF;
	
	IF LCP.Section[i].Sust.ShortContact2_close = TRUE AND LCP.Section[i].Sust.UnshortContact2_close = FALSE 
		THEN
			LCP.Section[i].Sust.ShortContact2Engaged := TRUE;
		ELSE
			LCP.Section[i].Sust.ShortContact2Engaged := FALSE;
	END_IF;
	
END_FOR;

//Formation
IF LCP.Section[4].Form.ShortContact1_close = TRUE AND LCP.Section[4].Form.UnshortContact1_close = FALSE
	THEN
		LCP.Section[4].Form.ShortContact1Engaged := TRUE;
	ELSE
		LCP.Section[4].Form.ShortContact1Engaged := FALSE; //might need to clarify on the NC of the short contacts.
END_IF;

IF LCP.Section[4].Form.ShortContact2_close = TRUE AND LCP.Section[4].Form.UnshortContact2_close = FALSE 
	THEN
		LCP.Section[4].Form.ShortContact2Engaged := TRUE;
	ELSE
		LCP.Section[4].Form.ShortContact2Engaged := FALSE; //might need to clarify on the NC of the short contacts.
END_IF;

// form trig short 
IF LCP.Section[4].Form.FormTrigShortContact_close = TRUE AND LCP.Section[4].Form.FormTrigUnShortContact_close = FALSE
	THEN
		LCP.Section[4].Form.FormTrigShortContactEngaged := TRUE;
	ELSE
		LCP.Section[4].Form.FormTrigShortContactEngaged := FALSE;
END_IF
// preform trig short 
IF LCP.Section[4].Form.PreFormTrigShortContact_close = TRUE AND LCP.Section[4].Form.PreFormTrigUnShortContact_close = FALSE
	THEN
		LCP.Section[4].Form.PreFormTrigShortContactEngaged := TRUE;
	ELSE
		LCP.Section[4].Form.PreFormTrigShortContactEngaged := FALSE;
END_IF

//short contacts unknown - This should have never happen
FOR i := 1 TO 3 BY 1 DO
	//Peak
	IF (LCP.Section[i].Peak.ShortContact1_close = TRUE AND LCP.Section[i].Peak.UnShortContact1_close = TRUE) OR 
 		(LCP.Section[i].Peak.ShortContact1_close = FALSE AND LCP.Section[i].Peak.UnShortContact1_close = FALSE)
		THEN
			LCP.Section[i].Peak.ShortContact1unknown := TRUE;
			ELSE
				LCP.Section[i].Peak.ShortContact1unknown := FALSE;
	END_IF;
	
	IF (LCP.Section[i].Peak.ShortContact2_close = TRUE AND LCP.Section[i].Peak.UnShortContact2_close = TRUE) OR 
 		(LCP.Section[i].Peak.ShortContact2_close = FALSE AND LCP.Section[i].Peak.UnShortContact2_close = FALSE)
		THEN
			LCP.Section[i].Peak.ShortContact2unknown := TRUE;
			ELSE
				LCP.Section[i].Peak.ShortContact2unknown := FALSE;
	END_IF;
	//Sust
	IF (LCP.Section[i].Sust.ShortContact1_close = TRUE AND LCP.Section[i].Sust.UnShortContact1_close = TRUE) OR 
 		(LCP.Section[i].Sust.ShortContact1_close = FALSE AND LCP.Section[i].Sust.UnShortContact1_close = FALSE)
		THEN
			LCP.Section[i].Sust.ShortContact1unknown := TRUE;
			ELSE
				LCP.Section[i].Sust.ShortContact1unknown := FALSE;
	END_IF;	
	
	IF (LCP.Section[i].Sust.ShortContact2_close = TRUE AND LCP.Section[i].Sust.UnShortContact2_close = TRUE) OR 
 		(LCP.Section[i].Sust.ShortContact2_close = FALSE AND LCP.Section[i].Sust.UnShortContact2_close = FALSE)
		THEN
			LCP.Section[i].Sust.ShortContact2unknown := TRUE;
			ELSE
				LCP.Section[i].Sust.ShortContact2unknown := FALSE;
	END_IF;	
	
END_FOR;

//Formation
IF (LCP.Section[4].Form.ShortContact1_close = TRUE AND LCP.Section[4].Form.UnShortContact1_close = TRUE) OR 
 	(LCP.Section[4].Form.ShortContact1_close = FALSE AND LCP.Section[4].Form.UnShortContact1_close = FALSE)
	THEN
		LCP.Section[4].Form.ShortContact1unknown := TRUE;
		ELSE
			LCP.Section[4].Form.ShortContact1unknown := FALSE;
END_IF;	
	
IF (LCP.Section[4].Form.ShortContact2_close = TRUE AND LCP.Section[4].Form.UnShortContact2_close = TRUE) OR 
 	(LCP.Section[4].Form.ShortContact2_close = FALSE AND LCP.Section[4].Form.UnShortContact2_close = FALSE)
	THEN
		LCP.Section[4].Form.ShortContact2unknown := TRUE;
		ELSE
			LCP.Section[4].Form.ShortContact2unknown := FALSE;
END_IF;	

IF (LCP.Section[4].Form.FormTrigUnshortContact_close = TRUE AND LCP.Section[4].Form.FormTrigUnshortContact_close = TRUE) OR 
	(LCP.Section[4].Form.FormTrigUnshortContact_close = FALSE AND LCP.Section[4].Form.FormTrigUnshortContact_close = FALSE)
	THEN 
		LCP.Section[4].Form.FormTrigShortContactUnknown := TRUE;
		ELSE
			LCP.Section[4].Form.FormTrigShortContactUnknown := FALSE;
END_IF;

IF (LCP.Section[4].Form.PreFormTrigShortContact_close = TRUE AND LCP.Section[4].Form.PreFormTrigUnShortContact_close = TRUE) OR
	(LCP.Section[4].Form.PreFormTrigShortContact_close = FALSE AND LCP.Section[4].Form.PreFormTrigUnShortContact_close = FALSE)
	THEN
		LCP.Section[4].Form.PreFormTrigShortContactUnknown := TRUE;
		ELSE
			LCP.Section[4].Form.PreFormTrigShortContactUnknown := FALSE;
END_IF;
	
// any short contact in unknown state?
IF LCP.Section[1].Peak.ShortContact1unknown = FALSE AND 
	LCP.Section[1].Peak.ShortContact2unknown = FALSE AND
	LCP.Section[2].Peak.ShortContact1unknown = FALSE AND
	LCP.Section[2].Peak.ShortContact2unknown = FALSE AND
	LCP.Section[3].Peak.ShortContact1unknown = FALSE AND
	LCP.Section[3].Peak.ShortContact2unknown = FALSE AND
	LCP.Section[1].Sust.ShortContact1unknown = FALSE AND
	LCP.Section[1].Sust.ShortContact2unknown = FALSE AND
	LCP.Section[2].Sust.ShortContact1unknown = FALSE AND 
	LCP.Section[2].Sust.ShortContact2unknown = FALSE AND
	LCP.Section[3].Sust.ShortContact1unknown = FALSE AND 
	LCP.Section[3].Sust.ShortContact2unknown = FALSE AND
	LCP.Section[4].Form.ShortContact1unknown = FALSE AND
	LCP.Section[4].Form.ShortContact2unknown = FALSE AND 
	LCP.Section[4].Form.FormTrigShortContactUnknown = FALSE AND //
	LCP.Section[4].Form.PreFormTrigShortContactUnknown = FALSE //
	THEN
		Permissives_DB.NoShortingUnknowns := TRUE;
	ELSE
		Permissives_DB.NoShortingUnknowns := FALSE;
END_IF;


//any short contact engaged

IF LCP.Section[1].Peak.ShortContact1Engaged = TRUE AND 
	LCP.Section[1].Peak.ShortContact2Engaged = TRUE AND
	LCP.Section[2].Peak.ShortContact1Engaged = TRUE AND
	LCP.Section[2].Peak.ShortContact2Engaged = TRUE AND
	LCP.Section[3].Peak.ShortContact1Engaged = TRUE AND
	LCP.Section[3].Peak.ShortContact2Engaged = TRUE AND
	LCP.Section[1].Sust.ShortContact1Engaged = TRUE AND
	LCP.Section[1].Sust.ShortContact2Engaged = TRUE AND
	LCP.Section[2].Sust.ShortContact1Engaged = TRUE AND 
	LCP.Section[2].Sust.ShortContact2Engaged = TRUE AND
	LCP.Section[3].Sust.ShortContact1Engaged = TRUE AND 
	LCP.Section[3].Sust.ShortContact2Engaged = TRUE AND
	LCP.Section[4].Form.ShortContact1Engaged = TRUE AND
	LCP.Section[4].Form.ShortContact2Engaged = TRUE AND 
	LCP.Section[4].Form.FormTrigShortContactEngaged = TRUE AND //
	LCP.Section[4].Form.PreFormTrigShortContactEngaged = TRUE //
	THEN
		Permissives_DB.AllShortContactEngaged := TRUE;
	ELSE 
		Permissives_DB.AllShortContactEngaged := FALSE;	
END_IF;

//All charger inhibited
IF (MCP_IO.Charger[1].inhibited = TRUE OR Recipe.PeakSupplyEN = FALSE) AND
	(MCP_IO.Charger[2].inhibited = TRUE OR Recipe.PeakSupplyEN = FALSE) AND
	(MCP_IO.Charger[3].inhibited = TRUE OR Recipe.PeakSupplyEN = FALSE) AND
	(MCP_IO.Charger[4].inhibited = TRUE OR Recipe.SustSupplyEN = FALSE) AND
	(MCP_IO.Charger[5].inhibited = TRUE OR Recipe.SustSupplyEN = FALSE) AND
	(MCP_IO.Charger[6].inhibited = TRUE OR Recipe.SustSupplyEN = FALSE) AND
	(MCP_IO.Charger[7].inhibited = TRUE OR Recipe.FormSupplyEN = FALSE) AND
	(MCP_IO.Charger[8].inhibited = TRUE OR Recipe.FormSupplyEN = FALSE) 
	THEN
		Permissives_DB.AllChargerInhibited := TRUE;
		ELSE
			Permissives_DB.AllChargerInhibited := FALSE;
END_IF;

//All charger HV ON
IF (MCP_IO.Charger[1].HV_isON = TRUE OR Recipe.PeakSupplyEN = FALSE) AND
	(MCP_IO.Charger[2].HV_isON = TRUE OR Recipe.PeakSupplyEN = FALSE) AND
	(MCP_IO.Charger[3].HV_isON = TRUE OR Recipe.PeakSupplyEN = FALSE) AND
	(MCP_IO.Charger[4].HV_isON = TRUE OR Recipe.SustSupplyEN = FALSE) AND
	(MCP_IO.Charger[5].HV_isON = TRUE OR Recipe.SustSupplyEN = FALSE) AND
	(MCP_IO.Charger[6].HV_isON = TRUE OR Recipe.SustSupplyEN = FALSE) AND
	(MCP_IO.Charger[7].HV_isON = TRUE OR Recipe.FormSupplyEN = FALSE) AND
	(MCP_IO.Charger[8].HV_isON = TRUE OR Recipe.FormSupplyEN = FALSE) AND
	(MCP_IO.GLS3_hvON = TRUE OR Recipe.PFormSupplyEN = FALSE)
	THEN
		Permissives_DB.AllChargerHVisON := TRUE;
		ELSE
			Permissives_DB.AllChargerHVisON := FALSE;
END_IF;

//peaking ch hv on
IF MCP_IO.Charger[1].HV_isON = TRUE AND 
	MCP_IO.Charger[2].HV_isON = TRUE AND 
	MCP_IO.Charger[3].HV_isON = TRUE 
	THEN
		Permissives_DB.AllPeakChargerHVisON := TRUE;
		ELSE
			Permissives_DB.AllPeakChargerHVisON := FALSE;
END_IF
//sustain ch hv on
IF MCP_IO.Charger[4].HV_isON = TRUE AND 
	MCP_IO.Charger[5].HV_isON = TRUE AND 
	MCP_IO.Charger[6].HV_isON = TRUE 
	THEN
		Permissives_DB.AllSustChargerHVisON := TRUE;
		ELSE
			Permissives_DB.AllSustChargerHVisON := FALSE;
END_IF
//Form ch hv on
IF MCP_IO.Charger[7].HV_isON = TRUE AND 
	MCP_IO.Charger[8].HV_isON = TRUE  
	THEN
		Permissives_DB.AllFormChargerHVisON := TRUE;
		ELSE
			Permissives_DB.AllFormChargerHVisON := FALSE;
END_IF
//peaking ch inhibit
IF MCP_IO.Charger[1].inhibited = TRUE AND 
	MCP_IO.Charger[2].inhibited = TRUE AND 
	MCP_IO.Charger[3].inhibited = TRUE 
	THEN
		Permissives_DB.AllPeakChargerInhibited := TRUE;
		ELSE
			Permissives_DB.AllPeakChargerInhibited := FALSE;
END_IF
//sust ch inhibit
IF MCP_IO.Charger[4].inhibited = TRUE AND 
	MCP_IO.Charger[5].inhibited = TRUE AND 
	MCP_IO.Charger[6].inhibited = TRUE 
	THEN
		Permissives_DB.AllSustChargerInhibited := TRUE;
		ELSE
			Permissives_DB.AllSustChargerInhibited := FALSE;
END_IF
//form ch inhibit
IF MCP_IO.Charger[7].inhibited = TRUE AND 
	MCP_IO.Charger[8].inhibited = TRUE
	THEN
		Permissives_DB.AllFormChargerInhibited := TRUE;
		ELSE
			Permissives_DB.AllFormChargerInhibited := FALSE;
END_IF

IF (MCP_IO.Charger[1].EndOfCharge = TRUE OR Recipe.PeakSupplyEN = FALSE) AND
	(MCP_IO.Charger[2].EndOfCharge = TRUE OR Recipe.PeakSupplyEN = FALSE) AND
	(MCP_IO.Charger[3].EndOfCharge = TRUE OR Recipe.PeakSupplyEN = FALSE) AND
	(MCP_IO.Charger[4].EndOfCharge = TRUE OR Recipe.SustsupplyEN = FALSE) AND
	(MCP_IO.Charger[5].EndOfCharge = TRUE OR Recipe.SustsupplyEN = FALSE) AND
	(MCP_IO.Charger[6].EndOfCharge = TRUE OR Recipe.SustsupplyEN = FALSE) AND
	(MCP_IO.Charger[7].EndOfCharge = TRUE OR Recipe.FormSupplyEN = FALSE) AND
	(MCP_IO.Charger[8].EndOfCharge = TRUE OR Recipe.FormSupplyEN = FALSE) 
	THEN 
		Permissives_DB.AllChargerEOC := TRUE;
		ELSE
			Permissives_DB.AllChargerEOC := FALSE;
END_IF

//all peaking charg
IF LCP.Section[1].Peak.ChargeRelay1_close = TRUE AND
	LCP.Section[1].Peak.ChargeRelay2_close = TRUE AND
	LCP.Section[2].Peak.ChargeRelay1_close = TRUE AND
	LCP.Section[2].Peak.ChargeRelay2_close = TRUE AND
	LCP.Section[3].Peak.ChargeRelay1_close = TRUE AND
	LCP.Section[3].Peak.ChargeRelay2_close = TRUE 
	THEN
		Permissives_DB.AllPeakChargeRlyClose := TRUE;
		ELSE
			Permissives_DB.AllPeakChargeRlyClose := FALSE;
END_IF

//all sust charge
IF LCP.Section[1].Sust.ChargeRelay1_close = TRUE AND
	LCP.Section[1].Sust.ChargeRelay2_close = TRUE AND
	LCP.Section[2].Sust.ChargeRelay1_close = TRUE AND
	LCP.Section[2].Sust.ChargeRelay2_close = TRUE AND
	LCP.Section[3].Sust.ChargeRelay1_close = TRUE AND
	LCP.Section[3].Sust.ChargeRelay2_close = TRUE 
	THEN
		Permissives_DB.AllSustChargeRlyClose := TRUE;
		ELSE
			Permissives_DB.AllSustChargeRlyClose := FALSE;
END_IF
//all form charge
IF	LCP.Section[4].Form.ChargeRelay1_close = TRUE AND
	LCP.Section[4].Form.ChargeRelay2_close = TRUE 
	THEN
		Permissives_DB.AllFormChargeRlyClose := TRUE;
		ELSE
			Permissives_DB.AllFormChargeRlyClose := FALSE;
END_IF

//all peak dump
IF LCP.Section[1].Peak.DumpRelay1_close = TRUE AND
	LCP.Section[1].Peak.DumpRelay2_close = TRUE AND
	LCP.Section[2].Peak.DumpRelay1_close = TRUE AND
	LCP.Section[2].Peak.DumpRelay2_close = TRUE AND
	LCP.Section[3].Peak.DumpRelay1_close = TRUE AND
	LCP.Section[3].Peak.DumpRelay2_close = TRUE 
	THEN
		Permissives_DB.AllPeakDumpRlyOpen := FALSE;
		ELSE
			Permissives_DB.AllPeakDumpRlyOpen := TRUE;
END_IF
//all sust dump
IF LCP.Section[1].Sust.DumpRelay1_close = TRUE AND
	LCP.Section[1].Sust.DumpRelay2_close = TRUE AND
	LCP.Section[2].Sust.DumpRelay1_close = TRUE AND
	LCP.Section[2].Sust.DumpRelay2_close = TRUE AND
	LCP.Section[3].Sust.DumpRelay1_close = TRUE AND
	LCP.Section[3].Sust.DumpRelay2_close = TRUE 
	THEN
		Permissives_DB.AllSustDumpRlyOpen := FALSE;
		ELSE
			Permissives_DB.AllSustDumpRlyOpen := TRUE;
END_IF
//all form dump
IF LCP.Section[4].Form.DumpRelay1_close = TRUE AND
	LCP.Section[4].Form.DumpRelay2_close = TRUE 
	THEN
		Permissives_DB.AllFormDumpRlyOpen := FALSE;
		ELSE
			Permissives_DB.AllFormDumpRlyOpen := TRUE;
END_IF
// GLS 1 & 2 can use raw input bit.

//section 1 charge
IF LCP.Section[1].Peak.ChargeRelay1_close = TRUE AND
	LCP.Section[1].Peak.ChargeRelay2_close = TRUE AND
	LCP.Section[1].Sust.ChargeRelay1_close = TRUE AND
	LCP.Section[1].Sust.ChargeRelay2_close = TRUE 
	THEN
		Permissives_DB.AllSection1ChargeRlyClose := TRUE;
		ELSE
			Permissives_DB.AllSection1ChargeRlyClose := FALSE;
END_IF;
//section 2 charge
IF LCP.Section[2].Peak.ChargeRelay1_close = TRUE AND
	LCP.Section[2].Peak.ChargeRelay2_close = TRUE AND
	LCP.Section[2].Sust.ChargeRelay1_close = TRUE AND
	LCP.Section[2].Sust.ChargeRelay2_close = TRUE 
	THEN
		Permissives_DB.AllSection2ChargeRlyClose := TRUE;
		ELSE
			Permissives_DB.AllSection2ChargeRlyClose := FALSE;
END_IF;
//section 3 charge
IF LCP.Section[3].Peak.ChargeRelay1_close = TRUE AND
	LCP.Section[3].Peak.ChargeRelay2_close = TRUE AND
	LCP.Section[3].Sust.ChargeRelay1_close = TRUE AND
	LCP.Section[3].Sust.ChargeRelay2_close = TRUE 
	THEN
		Permissives_DB.AllSection3ChargeRlyClose := TRUE;
		ELSE
			Permissives_DB.AllSection3ChargeRlyClose := FALSE;
END_IF;
//section 4 charge
IF	LCP.Section[4].Form.ChargeRelay1_close = TRUE AND
	LCP.Section[4].Form.ChargeRelay2_close = TRUE AND						
	LCP.Section[4].Form.PreFormChargeRly_close = TRUE AND
	LCP.Section[4].Form.FormTrigChargeRly_close = TRUE AND
	LCP.Section[4].Form.PreFormTrigChargeRly_close = TRUE
	THEN
		Permissives_DB.AllSection4ChargeRlyClose := TRUE;
		ELSE
			Permissives_DB.AllSection4ChargeRlyClose := FALSE;
END_IF
	
//All charge relay close
IF ((LCP.Section[1].Peak.ChargeRelay1_close = TRUE OR Recipe.PeakSupplyEN = FALSE)AND
	(LCP.Section[1].Peak.ChargeRelay2_close = TRUE OR Recipe.PeakSupplyEN = FALSE)AND
	(LCP.Section[1].Sust.ChargeRelay1_close = TRUE OR Recipe.SustSupplyEN = FALSE)AND
	(LCP.Section[1].Sust.ChargeRelay2_close = TRUE OR Recipe.SustSupplyEN = FALSE)AND
	(LCP.Section[2].Peak.ChargeRelay1_close = TRUE OR Recipe.PeakSupplyEN = FALSE)AND
	(LCP.Section[2].Peak.ChargeRelay2_close = TRUE OR Recipe.PeakSupplyEN = FALSE)AND
	(LCP.Section[2].Sust.ChargeRelay1_close = TRUE OR Recipe.SustSupplyEN = FALSE)AND
	(LCP.Section[2].Sust.ChargeRelay2_close = TRUE OR Recipe.SustSupplyEN = FALSE)AND
	(LCP.Section[3].Peak.ChargeRelay1_close = TRUE OR Recipe.PeakSupplyEN = FALSE)AND
	(LCP.Section[3].Peak.ChargeRelay2_close = TRUE OR Recipe.PeakSupplyEN = FALSE)AND
	(LCP.Section[3].Sust.ChargeRelay1_close = TRUE OR Recipe.SustSupplyEN = FALSE)AND
	(LCP.Section[3].Sust.ChargeRelay2_close = TRUE OR Recipe.SustSupplyEN = FALSE)AND
	
	(LCP.Section[4].Form.ChargeRelay1_close = TRUE OR Recipe.FormSupplyEN = FALSE)AND
	(LCP.Section[4].Form.ChargeRelay2_close = TRUE OR Recipe.FormSupplyEN = FALSE)AND						
	(LCP.Section[4].Form.PreFormChargeRly_close = TRUE OR Recipe.PFormSupplyEN = FALSE)AND
	(LCP.Section[4].Form.FormTrigChargeRly_close = TRUE  OR Recipe.FormSupplyEN = FALSE)AND
	(LCP.Section[4].Form.PreFormTrigChargeRly_close = TRUE OR Recipe.PFormSupplyEN = FALSE)) OR HMI_DB.AllChargeRelayCloseBP = TRUE //admin bypass 
	THEN
		Permissives_DB.AllChargeRelaysClosed := TRUE;
	ELSE
		Permissives_DB.AllChargeRelaysClosed := FALSE;
END_IF;

//section 1 dump
IF LCP.Section[1].Peak.DumpRelay1_close = FALSE AND
	LCP.Section[1].Peak.DumpRelay2_close = FALSE AND
	LCP.Section[1].Sust.DumpRelay1_close = FALSE AND
	LCP.Section[1].Sust.DumpRelay2_close = FALSE
	THEN
		Permissives_DB.AllSection1DumpRlyOpen := TRUE;
		ELSE
			Permissives_DB.AllSection1DumpRlyOpen := FALSE;
END_IF
//section 2 dump
IF LCP.Section[2].Peak.DumpRelay1_close = FALSE AND
	LCP.Section[2].Peak.DumpRelay2_close = FALSE AND
	LCP.Section[2].Sust.DumpRelay1_close = FALSE AND
	LCP.Section[2].Sust.DumpRelay2_close = FALSE
	THEN
		Permissives_DB.AllSection2DumpRlyOpen := TRUE;
		ELSE
			Permissives_DB.AllSection2DumpRlyOpen := FALSE;
END_IF
//section 3 dump
IF LCP.Section[3].Peak.DumpRelay1_close = FALSE AND
	LCP.Section[3].Peak.DumpRelay2_close = FALSE AND
	LCP.Section[3].Sust.DumpRelay1_close = FALSE AND
	LCP.Section[3].Sust.DumpRelay2_close = FALSE
	THEN
		Permissives_DB.AllSection3DumpRlyOpen := TRUE;
		ELSE
			Permissives_DB.AllSection3DumpRlyOpen := FALSE;
END_IF
//section 4 dump
IF 	LCP.Section[4].Form.DumpRelay1_close = FALSE AND
	LCP.Section[4].Form.DumpRelay2_close = FALSE AND						
	LCP.Section[4].Form.PreFormDumpRly_close = FALSE AND
	LCP.Section[4].Form.FormTrigDumpRly1_close = FALSE AND
	LCP.Section[4].Form.PreFormTrigDumpRly1_close = FALSE
	THEN
		Permissives_DB.AllSection4DumpRlyOpen := TRUE;
		ELSE
			Permissives_DB.AllSection4DumpRlyOpen := FALSE;
END_IF

//All Dump relays open  ******
IF (LCP.Section[1].Peak.DumpRelay1_close = FALSE AND
	LCP.Section[1].Peak.DumpRelay2_close = FALSE AND
	LCP.Section[1].Sust.DumpRelay1_close = FALSE AND
	LCP.Section[1].Sust.DumpRelay2_close = FALSE AND
	LCP.Section[2].Peak.DumpRelay1_close = FALSE AND
	LCP.Section[2].Peak.DumpRelay2_close = FALSE AND
	LCP.Section[2].Sust.DumpRelay1_close = FALSE AND
	LCP.Section[2].Sust.DumpRelay2_close = FALSE AND
	LCP.Section[3].Peak.DumpRelay1_close = FALSE AND
	LCP.Section[3].Peak.DumpRelay2_close = FALSE AND
	LCP.Section[3].Sust.DumpRelay1_close = FALSE AND
	LCP.Section[3].Sust.DumpRelay2_close = FALSE AND
	
	LCP.Section[4].Form.DumpRelay1_close = FALSE AND
	LCP.Section[4].Form.DumpRelay2_close = FALSE AND						
	LCP.Section[4].Form.PreFormDumpRly_close = FALSE AND
	LCP.Section[4].Form.FormTrigDumpRly1_close = FALSE AND
	LCP.Section[4].Form.PreFormTrigDumpRly1_close = FALSE) OR HMI_DB.AllDumpRelaysOpenBP = TRUE //admin bypass 
	THEN
		Permissives_DB.AllDumpRelaysOpen := TRUE;
	ELSE
		Permissives_DB.AllDumpRelaysOpen := FALSE;
END_IF;
//check for cap voltage for fully discharged
FOR i := 1 TO 3 BY 1 DO
	//peak
	FOR k := 1 TO 10 BY 1 DO
		IF LCP.Section[i].Peak.Cap[k].voltageFeedback <= 10 THEN 
			LCP.Section[i].Peak.Cap[k].CapDischaged := TRUE;
			ELSE
				LCP.Section[i].Peak.Cap[k].CapDischaged := FALSE;
		END_IF;
		//check for cap fully charged*************************
		IF LCP.Section[i].Peak.Cap[k].voltageFeedback >= Setpoints.TDKLoad[i].RequiredChargedV THEN 
			LCP.Section[i].Peak.Cap[k].CapfullyCharged := TRUE;
			ELSE
				LCP.Section[i].Peak.Cap[k].CapfullyCharged := FALSE;
		END_IF;
	END_FOR;
	//sus
	IF LCP.Section[i].Sust.Cap[1].voltageFeedback <= 10 THEN
		LCP.Section[i].Sust.Cap[1].CapDischaged := TRUE;
		ELSE
			LCP.Section[i].Sust.Cap[1].CapDischaged := FALSE;
	END_IF;
	//check fo cap fully charged
	IF LCP.Section[i].Sust.Cap[1].voltageFeedback >= Setpoints.TDKLoad[i+3].RequiredChargedV THEN
		LCP.Section[i].Sust.Cap[1].CapfullyCharged := TRUE;
		ELSE
			LCP.Section[i].Sust.Cap[1].CapfullyCharged := FALSE;
	END_IF;
	
	IF LCP.Section[i].Sust.Cap[2].voltageFeedback <= 10 THEN
		LCP.Section[i].Sust.Cap[2].CapDischaged := TRUE;
		ELSE
			LCP.Section[i].Sust.Cap[2].CapDischaged := FALSE;
	END_IF;
	//check for cap fully charged
	IF LCP.Section[i].Sust.Cap[2].voltageFeedback >= Setpoints.TDKLoad[i+3].RequiredChargedV THEN
		LCP.Section[i].Sust.Cap[2].CapfullyCharged := TRUE;
		ELSE
			LCP.Section[i].Sust.Cap[2].CapfullyCharged := FALSE;
	END_IF;
END_FOR;
// form
FOR m := 1 TO 12 BY 1 DO
	IF LCP.Section[4].Form.Cap[m].voltageFeedback <= 10 THEN
		LCP.Section[4].Form.Cap[m].CapDischaged := TRUE;
		ELSE
			LCP.Section[4].Form.Cap[m].CapDischaged := FALSE;
	END_IF;
END_FOR;

//check for cap fully charged
FOR n := 1 TO 6 BY 1 DO 
	IF LCP.Section[4].Form.Cap[n].voltageFeedback >= Setpoints.TDKLoad[7].RequiredChargedV THEN
		LCP.Section[4].Form.Cap[n].CapfullyCharged := TRUE;
		ELSE
			LCP.Section[4].Form.Cap[n].CapfullyCharged := FALSE;
	END_IF;		
END_FOR

FOR p := 7 TO 12 BY 1 DO 
	IF LCP.Section[4].Form.Cap[p].voltageFeedback >= Setpoints.TDKLoad[8].RequiredChargedV THEN
		LCP.Section[4].Form.Cap[p].CapfullyCharged := TRUE;
		ELSE
			LCP.Section[4].Form.Cap[p].CapfullyCharged := FALSE;
	END_IF;		
END_FOR

//preform
IF LCP.Section[4].PreFormCapVoltageFeedback <= 10 THEN
	LCP.Section[4].PreFormCapDischarged := TRUE;
	ELSE
		LCP.Section[4].PreFormCapDischarged := FALSE;
END_IF

//preform
IF LCP.Section[4].PreFormCapVoltageFeedback >= Setpoints.GLSLoad.RequiredChargedV THEN
	LCP.Section[4].PreFormCapFullyChaged := TRUE;
	ELSE
		LCP.Section[4].PreFormCapFullyChaged := FALSE;
END_IF


//all caps discharge condition
FOR i := 1 TO 3 BY 1 DO
	IF LCP.Section[i].Peak.Cap[1].CapDischaged = TRUE AND
		LCP.Section[i].Peak.Cap[2].CapDischaged = TRUE AND
		LCP.Section[i].Peak.Cap[3].CapDischaged = TRUE AND
		LCP.Section[i].Peak.Cap[4].CapDischaged = TRUE AND
		LCP.Section[i].Peak.Cap[5].CapDischaged = TRUE AND
		LCP.Section[i].Peak.Cap[6].CapDischaged = TRUE AND
		LCP.Section[i].Peak.Cap[7].CapDischaged = TRUE AND
		LCP.Section[i].Peak.Cap[8].CapDischaged = TRUE AND
		LCP.Section[i].Peak.Cap[9].CapDischaged = TRUE AND
		LCP.Section[i].Peak.Cap[10].CapDischaged = TRUE AND
		LCP.Section[i].Sust.Cap[1].CapDischaged = TRUE AND
		LCP.Section[i].Sust.Cap[2].CapDischaged = TRUE
		THEN
			LCP.Section[i].AllCapsDischarged := TRUE; 
		ELSE
			LCP.Section[i].AllCapsDischarged := FALSE; 
	END_IF;
	
	//all caps fully charged 
	IF LCP.Section[i].Peak.Cap[1].CapFullyCharged = TRUE AND
		LCP.Section[i].Peak.Cap[2].CapFullyCharged = TRUE AND
		LCP.Section[i].Peak.Cap[3].CapFullyCharged = TRUE AND
		LCP.Section[i].Peak.Cap[4].CapFullyCharged = TRUE AND
		LCP.Section[i].Peak.Cap[5].CapFullyCharged = TRUE AND
		LCP.Section[i].Peak.Cap[6].CapFullyCharged = TRUE AND
		LCP.Section[i].Peak.Cap[7].CapFullyCharged = TRUE AND
		LCP.Section[i].Peak.Cap[8].CapFullyCharged = TRUE AND
		LCP.Section[i].Peak.Cap[9].CapFullyCharged = TRUE AND
		LCP.Section[i].Peak.Cap[10].CapFullyCharged = TRUE AND
		LCP.Section[i].Sust.Cap[1].CapFullyCharged = TRUE AND
		LCP.Section[i].Sust.Cap[2].CapFullyCharged = TRUE
		THEN
			LCP.Section[i].AllCapsFullyCharged := TRUE;
		ELSE
			LCP.Section[i].AllCapsFullyCharged := FALSE;
	END_IF
END_FOR
//form caps 
IF LCP.Section[4].Form.Cap[1].CapDischaged = TRUE AND
	LCP.Section[4].Form.Cap[2].CapDischaged = TRUE AND
	LCP.Section[4].Form.Cap[3].CapDischaged = TRUE AND
	LCP.Section[4].Form.Cap[4].CapDischaged = TRUE AND
	LCP.Section[4].Form.Cap[5].CapDischaged = TRUE AND
	LCP.Section[4].Form.Cap[6].CapDischaged = TRUE AND
	LCP.Section[4].Form.Cap[7].CapDischaged = TRUE AND
	LCP.Section[4].Form.Cap[8].CapDischaged = TRUE AND
	LCP.Section[4].Form.Cap[9].CapDischaged = TRUE AND
	LCP.Section[4].Form.Cap[10].CapDischaged = TRUE AND
	LCP.Section[4].Form.Cap[11].CapDischaged = TRUE AND
	LCP.Section[4].Form.Cap[12].CapDischaged = TRUE AND 
	LCP.Section[4].PreFormCapDischarged = TRUE
	THEN 
		LCP.Section[4].AllCapsDischarged := TRUE;
	ELSE
		LCP.Section[4].AllCapsDischarged := FALSE;	
END_IF
//checking for caps fully charged
IF LCP.Section[4].Form.Cap[1].CapFullyCharged = TRUE AND
	LCP.Section[4].Form.Cap[2].CapFullyCharged = TRUE AND
	LCP.Section[4].Form.Cap[3].CapFullyCharged = TRUE AND
	LCP.Section[4].Form.Cap[4].CapFullyCharged = TRUE AND
	LCP.Section[4].Form.Cap[5].CapFullyCharged = TRUE AND
	LCP.Section[4].Form.Cap[6].CapFullyCharged = TRUE AND
	LCP.Section[4].Form.Cap[7].CapFullyCharged = TRUE AND
	LCP.Section[4].Form.Cap[8].CapFullyCharged = TRUE AND
	LCP.Section[4].Form.Cap[9].CapFullyCharged = TRUE AND
	LCP.Section[4].Form.Cap[10].CapFullyCharged = TRUE AND
	LCP.Section[4].Form.Cap[11].CapFullyCharged = TRUE AND
	LCP.Section[4].Form.Cap[12].CapFullyCharged = TRUE AND
	LCP.Section[4].PreFormCapFullyChaged = TRUE
	THEN
		LCP.Section[4].AllCapsFullyCharged := TRUE;
	ELSE
		LCP.Section[4].AllCapsFullyCharged := FALSE;
END_IF

//all capps fully charged
IF LCP.Section[1].AllCapsFullyCharged = TRUE AND
	LCP.Section[2].AllCapsFullyCharged = TRUE AND
	LCP.Section[3].AllCapsFullyCharged = TRUE AND
	LCP.Section[4].AllCapsFullyCharged = TRUE 
	THEN
		Permissives_DB.AllSectCapsFullyCharged := TRUE;
	ELSE
		Permissives_DB.AllSectCapsFullyCharged := FALSE;
END_IF

IF LCP.Section[1].AllCapsDischarged = TRUE AND
	LCP.Section[2].AllCapsDischarged = TRUE AND
	LCP.Section[3].AllCapsDischarged = TRUE AND
	LCP.Section[4].AllCapsDischarged = TRUE 
	THEN 
		Permissives_DB.AllSectCapsDischarged := TRUE;
	ELSE
		Permissives_DB.AllSectCapsDischarged := FALSE;
END_IF


//no loss in interlock pneumatic pressure

IF (LCP.Section[1].LossPneumaticPressure = FALSE AND
	LCP.Section[2].LossPneumaticPressure = FALSE AND
	LCP.Section[3].LossPneumaticPressure = FALSE AND
	LCP.Section[4].LossPneumaticPressure = FALSE) OR HMI_DB.InterlockPressureLossBP = TRUE 
	THEN
		Permissives_DB.NoInterlockPressureLoss := TRUE;
		ELSE
			Permissives_DB.NoInterlockPressureLoss := FALSE;
END_IF;
	
IF (Permissives_DB.NoShortingUnknowns = TRUE AND
	Trips_DB.AllDCpsuOK = TRUE AND
	Trips_DB.CageEStopCircuitBroken = FALSE AND
	Trips_DB.AnyChargerOverTemp = FALSE AND
	Trips_DB.AnyEstopPressed = FALSE AND
	Trips_DB.AnyChargerInterlockOpen = FALSE AND
	Permissives_DB.NoInterlockPressureLoss = TRUE) OR HMI_DB.SafetyOKBP = TRUE // admin bypass 
	THEN
		Permissives_DB.SafetyOK := TRUE;
		ELSE
			Permissives_DB.SafetyOK := FALSE;
END_IF;

IF i > 3 THEN
	i := 1;
END_IF;

IF j > 8 THEN
	j := 1;
END_IF;

IF k > 10 THEN
	k := 1;
END_IF;

IF m > 12 THEN
	m := 1;
END_IF;

IF n > 6 THEN
	n := 1;
END_IF;

IF p > 12 THEN
	p := 7;
END_IF;

END_PROGRAM

// ---- POUs/Trips.TcPOU
PROGRAM Trips
VAR
	bTest							: BOOL;
	//delay2s : Delay2s;
	evtLogger						: FB_TcEventLogger;
	
	ACintLockRlyFaultDelay_PT		: TIME := T#2S;
	DumpRlyFaultDelay_PT			: TIME := T#2S;
	//DumpRly2FaultDelay_PT			: TIME := T#2S;
	ChrgRlyFaultDelay_PT			: TIME := T#1S;
	
	LiftMachineGNDFaultTON			: TON;
	LiftMachineGNDFaultPT			: TIME := T#2000MS;
	
	GeneralFaultDelayPT				: TIME := T#500MS;
	
	stControl						: ST_Control;
	
	i : INT := 1;  //charger 1-8
	j : INT := 1; //section 1-3
	k : INT := 1; //section 1-4, might not need 
END_VAR


//MCP Input Trips
IF MCP_IO.MasterStopPB_Pressed = TRUE THEN
	Trips_DB.MasterStopPBPressed := TRUE;	
END_IF;

IF MCP_IO.CageEstopCircuitOK = FALSE THEN
	Trips_DB.CageEStopCircuitBroken := TRUE; 
END_IF;

IF MCP_IO.RemoteModeSelected = FALSE THEN
	Trips_DB.LocalModeSelected := TRUE; //may not be a trip
	ELSE
		Trips_DB.LocalModeSelected := FALSE;
END_IF;

IF MCP_IO.PSU1_DCOK = FALSE THEN
	Trips_DB.MCPLossDCpower := TRUE; 
END_IF;

IF (MCP_IO.LiftMachineGND = TRUE AND MCP_IO.MachineGNDrlyOpen = FALSE) OR 
	(MCP_IO.LiftMachineGND = FALSE AND MCP_IO.MachineGNDrlyOpen = TRUE)
	THEN
		//delay
		LiftMachineGNDFaultTON (IN := TRUE, PT := LiftMachineGNDFaultPT);
		IF LiftMachineGNDFaultTON.Q = TRUE THEN
			Trips_DB.MachineGNDrlyFailed := TRUE;
			LiftMachineGNDFaultTON (IN := FALSE);
		END_IF
	ELSE
		LiftMachineGNDFaultTON (IN := FALSE);
END_IF

FOR i := 1 TO 8 BY 1 DO
	//check for loss inhibit

	IF (MCP_IO.Charger[i].inhibit = TRUE AND MCP_IO.Charger[i].inhibited = FALSE) OR 
		(MCP_IO.Charger[i].inhibit = FALSE AND MCP_IO.Charger[i].inhibited = TRUE)
		THEN
			MCP_IO.Charger[i].LossInhibitTON (IN := TRUE, PT := GeneralFaultDelayPT);
			IF MCP_IO.Charger[i].LossInhibitTON.Q = TRUE THEN 
				MCP_IO.Charger[i].LossInhibit := TRUE; //for alarms and not an actual trip
				MCP_IO.Charger[i].LossInhibitTON (IN := FALSE);
			END_IF
		ELSE
			MCP_IO.Charger[i].LossInhibit := FALSE;
			MCP_IO.Charger[i].LossInhibitTON (IN := FALSE);
	END_IF
	//check for loss HV on signal
	IF MCP_IO.Charger[i].HV_ON = TRUE AND MCP_IO.Charger[i].HV_isON = FALSE 
		THEN
			MCP_IO.Charger[i].LossHVON_TON (IN := TRUE, PT := GeneralFaultDelayPT);
			IF MCP_IO.Charger[i].LossHVON_TON.Q = TRUE THEN
				MCP_IO.Charger[i].LossHVON := TRUE; //for alarms and not an actual trip
				MCP_IO.Charger[i].LossHVON_TON (IN := FALSE);
			END_IF
		ELSE
			MCP_IO.Charger[i].LossHVON := FALSE;
			MCP_IO.Charger[i].LossHVON_TON (IN := FALSE);
	END_IF
	//any loss inhibit signal and hv on signal
	IF MCP_IO.Charger[i].LossInhibit = TRUE THEN 
		Trips_DB.AnyLossInhibitSignal := TRUE;
	END_IF

END_FOR;

IF ((MCP_IO.Charger[1].LossHVON = TRUE AND Recipe.PeakSupplyEN = TRUE) OR
	(MCP_IO.Charger[2].LossHVON = TRUE AND Recipe.PeakSupplyEN = TRUE) OR
	(MCP_IO.Charger[3].LossHVON = TRUE AND Recipe.PeakSupplyEN = TRUE) OR
	(MCP_IO.Charger[4].LossHVON = TRUE AND Recipe.SustSupplyEN = TRUE) OR
	(MCP_IO.Charger[5].LossHVON = TRUE AND Recipe.SustSupplyEN = TRUE) OR
	(MCP_IO.Charger[6].LossHVON = TRUE AND Recipe.SustSupplyEN = TRUE) OR
	(MCP_IO.Charger[7].LossHVON = TRUE AND Recipe.FormSupplyEN = TRUE) OR
	(MCP_IO.Charger[8].LossHVON = TRUE AND Recipe.FormSupplyEN = TRUE)) AND HMI_DB.LossHVsignalBP = FALSE 
THEN
	Trips_DB.AnyLossHVONsignal := TRUE;
END_IF


// mapping pnumatic and dc power to trips
FOR k := 1 TO 4 BY 1 DO
	Trips_DB.Section[k].LossPneumaticPressure := LCP.Section[k].LossPneumaticPressure;
	Trips_DB.Section[k].LossDCPower := NOT LCP.Section[k].PSU1_DCOK;
END_FOR;


//any charge relay fail
IF Trips_DB.Section[1].Peak.ChargeRelay1_Failed = TRUE OR
	Trips_DB.Section[1].Peak.ChargeRelay2_Failed = TRUE OR
	Trips_DB.Section[1].Sust.ChargeRelay1_Failed = TRUE OR
	Trips_DB.Section[1].Sust.ChargeRelay2_Failed = TRUE OR
	Trips_DB.Section[2].Peak.ChargeRelay1_Failed = TRUE OR
	Trips_DB.Section[2].Peak.ChargeRelay2_Failed = TRUE OR
	Trips_DB.Section[2].Sust.ChargeRelay1_Failed = TRUE OR
	Trips_DB.Section[2].Sust.ChargeRelay2_Failed = TRUE OR
	Trips_DB.Section[3].Peak.ChargeRelay1_Failed = TRUE OR
	Trips_DB.Section[3].Peak.ChargeRelay2_Failed = TRUE OR
	Trips_DB.Section[3].Sust.ChargeRelay1_Failed = TRUE OR
	Trips_DB.Section[3].Sust.ChargeRelay2_Failed = TRUE OR
	Trips_DB.Section[4].Form.ChargeRelay1_Failed = TRUE OR 
	Trips_DB.Section[4].Form.ChargeRelay2_Failed = TRUE OR 
	Trips_DB.Section[4].Form.PreFormChrgRlyFailed = TRUE OR 
	Trips_DB.Section[4].Form.FormTrigChrgRlyFailed = TRUE OR
	Trips_DB.Section[4].Form.PreFormTrigChrgRlyFailed = TRUE		
	THEN 
		Trips_DB.AnyChargeRlyFail := TRUE;
	ELSE
		Trips_DB.AnyChargeRlyFail := FALSE;
END_IF;

//any dump relay fail
IF Trips_DB.Section[1].Peak.DumpRelay1_Failed = TRUE OR
	Trips_DB.Section[1].Peak.DumpRelay2_Failed = TRUE OR
	Trips_DB.Section[1].Sust.DumpRelay1_Failed = TRUE OR
	Trips_DB.Section[1].Sust.DumpRelay2_Failed = TRUE OR
	Trips_DB.Section[2].Peak.DumpRelay1_Failed = TRUE OR
	Trips_DB.Section[2].Peak.DumpRelay2_Failed = TRUE OR
	Trips_DB.Section[2].Sust.DumpRelay1_Failed = TRUE OR
	Trips_DB.Section[2].Sust.DumpRelay2_Failed = TRUE OR
	Trips_DB.Section[3].Peak.DumpRelay1_Failed = TRUE OR
	Trips_DB.Section[3].Peak.DumpRelay2_Failed = TRUE OR
	Trips_DB.Section[3].Sust.DumpRelay1_Failed = TRUE OR
	Trips_DB.Section[3].Sust.DumpRelay2_Failed = TRUE OR
	Trips_DB.Section[4].Form.DumpRelay1_Failed = TRUE OR 
	Trips_DB.Section[4].Form.DumpRelay2_Failed = TRUE OR 
	Trips_DB.Section[4].Form.PreFormDumpRlyFailed = TRUE OR 
	Trips_DB.Section[4].Form.FormTrigDumpRly1Failed = TRUE OR
	Trips_DB.Section[4].Form.PreFormTrigDumpRly1Failed = TRUE		
	THEN 
		Trips_DB.AnyDumpRlyFail := TRUE;
	ELSE
		Trips_DB.AnyDumpRlyFail := FALSE;
END_IF;

//if relays failed, chargers faulted, loss pneumatic pressure, or loss dc power then 
//Trips_DB.Section[j].SystemTripped := TRUE;

//system trip 
//section 1-3
FOR j := 1 TO 3 BY 1 DO
	IF Trips_DB.Section[j].LossDCPower = TRUE OR 
		Trips_DB.Section[j].LossPneumaticPressure = TRUE OR
		Trips_DB.Section[j].Peak.ChargeRelay1_Failed = TRUE OR
		Trips_DB.Section[j].Peak.ChargeRelay2_Failed = TRUE OR
		Trips_DB.Section[j].Peak.DumpRelay1_Failed = TRUE OR
		Trips_DB.Section[j].Peak.DumpRelay2_Failed = TRUE OR
		Trips_DB.Section[j].Sust.ChargeRelay1_Failed = TRUE OR
		Trips_DB.Section[j].Sust.ChargeRelay2_Failed = TRUE OR
		Trips_DB.Section[j].Sust.DumpRelay1_Failed = TRUE OR
		Trips_DB.Section[j].Sust.DumpRelay2_Failed = TRUE OR
		// shorted when not supposed to ?
		LCP.Section[j].Peak.ShortContact1unknown = TRUE OR // might need to  test it.  
		LCP.Section[j].Peak.ShortContact2unknown = TRUE 
		THEN
			Trips_DB.Section[j].SystemTripped := TRUE;
	END_IF;
END_FOR;

//formation
IF Trips_DB.Section[4].LossDCPower = TRUE OR 
	Trips_DB.Section[4].LossPneumaticPressure = TRUE OR
	Trips_DB.Section[4].Form.ChargeRelay1_Failed = TRUE OR
	Trips_DB.Section[4].Form.ChargeRelay2_Failed = TRUE OR
	Trips_DB.Section[4].Form.DumpRelay1_Failed = TRUE OR
	Trips_DB.Section[4].Form.DumpRelay2_Failed = TRUE OR
	Trips_DB.Section[4].Form.PreFormChrgRlyFailed = TRUE OR
	Trips_DB.Section[4].Form.FormTrigChrgRlyFailed = TRUE OR
	Trips_DB.Section[4].Form.PreFormTrigChrgRlyFailed = TRUE OR
	Trips_DB.Section[4].Form.PreFormDumpRlyFailed = TRUE OR
	Trips_DB.Section[4].Form.FormTrigDumpRly1Failed = TRUE OR
	Trips_DB.Section[4].Form.PreFormTrigDumpRly1Failed = TRUE OR 
	LCP.Section[4].Form.ShortContact1unknown = TRUE OR //might need to remove, might be too sensitive
	LCP.Section[4].Form.ShortContact2unknown = TRUE OR 
	LCP.Section[4].Form.FormTrigShortContactUnknown = TRUE OR 
	LCP.Section[4].Form.PreFormTrigShortContactUnknown = TRUE
	THEN
		Trips_DB.Section[4].SystemTripped := TRUE;
END_IF;


//Charger faults
FOR i := 1 TO 8 BY 1 DO
	//OVERTEMP 
	IF MCP_IO.Charger[i].OverTemp = TRUE THEN
		Trips_DB.AnyChargerOverTemp := TRUE;  
	END_IF;
	//Load faults
	IF MCP_IO.Charger[i].LoadFaulted = TRUE THEN
		Trips_DB.AnyChargerLoadFault := TRUE;  
	END_IF;
	//Interlock Open
	IF MCP_IO.Charger[i].InterlockOpen = TRUE THEN
		Trips_DB.AnyChargerInterlockOpen := TRUE;  
	END_IF;
	
END_FOR;

//Charger summary faults
FOR i := 1 TO 8 BY 1 DO
	IF MCP_IO.Charger[i].SummaryFaulted = TRUE THEN
		Trips_DB.AnyChargerFaulted := TRUE;  
	END_IF;
END_FOR;

//MCP trip
IF Trips_DB.AnyChargerFaulted = TRUE OR 
	Trips_DB.MasterStopPBPressed = TRUE OR
	Trips_DB.CageEStopCircuitBroken = TRUE OR
	Trips_DB.MCPLossDCpower = TRUE 
	THEN
		Trips_DB.MCPsystemTripped := TRUE;
END_IF


//*******************E-Stop Trips
IF MCP_IO.MasterStopPB_Pressed = TRUE OR MCP_IO.CageEstopCircuitOK THEN
	Trips_DB.AnyEstopPressed := TRUE;  
END_IF;	

//*********************DC PSU
IF (MCP_IO.PSU1_DCOK = TRUE AND 
	LCP.Section[1].PSU1_DCOK = TRUE AND
	LCP.Section[2].PSU1_DCOK = TRUE AND
	LCP.Section[3].PSU1_DCOK = TRUE AND
	LCP.Section[4].PSU1_DCOK = TRUE) OR HMI_DB.AlldcPSUokBP = TRUE //admin bypass 
	THEN
		TRIPS_DB.AllDCpsuOK := TRUE;
	ELSE 
		TRIPS_DB.AllDCpsuOK := FALSE;
END_IF;

//Relay faults***************************************
//section 1 - 3
FOR j := 1 TO 3 BY 1 DO
	//Peak Charge rly1
		//fail to close
	IF LCP.Section[j].Peak.CloseChargeRelay1 = TRUE AND LCP.Section[j].Peak.ChargeRelay1_close = FALSE THEN 
		//start timer
		Trips_DB.Section[j].Peak.ChrgRly1FaultDelay_TON (IN:= TRUE, PT := ChrgRlyFaultDelay_PT);
		
		IF Trips_DB.Section[j].Peak.ChrgRly1FaultDelay_TON.Q = TRUE THEN 
			Trips_DB.Section[j].Peak.ChargeRelay1_FailtoClose := TRUE; 
			Trips_DB.Section[j].Peak.ChrgRly1FaultDelay_TON (IN:= FALSE);
		END_IF;
	ELSE
		Trips_DB.Section[j].Peak.ChrgRly1FaultDelay_TON (IN:= FALSE);
	END_IF;

		//fail to open
	IF LCP.Section[j].Peak.CloseChargeRelay1 = FALSE AND LCP.Section[j].Peak.ChargeRelay1_close = TRUE THEN 
		//start timer
		Trips_DB.Section[j].Peak.ChrgRly1FaultDelay_TON (IN:= TRUE, PT := ChrgRlyFaultDelay_PT);
		
		IF Trips_DB.Section[j].Peak.ChrgRly1FaultDelay_TON.Q = TRUE THEN 
			Trips_DB.Section[j].Peak.ChargeRelay1_FailtoOpen := TRUE; 
			Trips_DB.Section[j].Peak.ChrgRly1FaultDelay_TON (IN:= FALSE);
		END_IF;
	ELSE
		Trips_DB.Section[j].Peak.ChrgRly1FaultDelay_TON (IN:= FALSE);
	END_IF;

	//Peak Charge rly2	
		//fail to close
	IF LCP.Section[j].Peak.CloseChargeRelay2 = TRUE AND LCP.Section[j].Peak.ChargeRelay2_close = FALSE THEN 
		//start timer
		Trips_DB.Section[j].Peak.ChrgRly2FaultDelay_TON (IN:= TRUE, PT := ChrgRlyFaultDelay_PT);
		
		IF Trips_DB.Section[j].Peak.ChrgRly2FaultDelay_TON.Q = TRUE THEN 
			Trips_DB.Section[j].Peak.ChargeRelay2_FailtoClose := TRUE; 
			Trips_DB.Section[j].Peak.ChrgRly2FaultDelay_TON (IN:= FALSE);
		END_IF;
	ELSE
		Trips_DB.Section[j].Peak.ChrgRly2FaultDelay_TON (IN:= FALSE);
	END_IF;
	
		//fail to open
	IF LCP.Section[j].Peak.CloseChargeRelay2 = FALSE AND LCP.Section[j].Peak.ChargeRelay2_close = TRUE THEN 
		//start timer
		Trips_DB.Section[j].Peak.ChrgRly2FaultDelay_TON (IN:= TRUE, PT := ChrgRlyFaultDelay_PT);
		
		IF Trips_DB.Section[j].Peak.ChrgRly2FaultDelay_TON.Q = TRUE THEN 
			Trips_DB.Section[j].Peak.ChargeRelay2_FailtoOpen := TRUE; 
			Trips_DB.Section[j].Peak.ChrgRly2FaultDelay_TON (IN:= FALSE);
		END_IF;
	ELSE
		Trips_DB.Section[j].Peak.ChrgRly2FaultDelay_TON (IN:= FALSE);
	END_IF;

	//Peak dump rly1
		//fail to open
	IF LCP.Section[j].Peak.OpenDumpRelay1 = TRUE AND LCP.Section[j].Peak.DumpRelay1_close = TRUE THEN 
		//start timer
		Trips_DB.Section[j].Peak.DumpRly1FaultDelay_TON (IN := TRUE, PT := DumpRlyFaultDelay_PT);

		IF Trips_DB.Section[j].Peak.DumpRly1FaultDelay_TON.Q = TRUE THEN 
			Trips_DB.Section[j].Peak.DumpRelay1_FailtoOpen := TRUE; 
			Trips_DB.Section[j].Peak.DumpRly1FaultDelay_TON (IN:= FALSE);
		END_IF; 
	ELSE
		Trips_DB.Section[j].Peak.DumpRly1FaultDelay_TON (IN:= FALSE);
	END_IF;

		//fail to close
	IF LCP.Section[j].Peak.OpenDumpRelay1 = FALSE AND LCP.Section[j].Peak.DumpRelay1_close = FALSE THEN 
		//start timer
		Trips_DB.Section[j].Peak.DumpRly1FaultDelay_TON (IN := TRUE, PT := DumpRlyFaultDelay_PT); 
		
		IF Trips_DB.Section[j].Peak.DumpRly1FaultDelay_TON.Q = TRUE THEN 
			Trips_DB.Section[j].Peak.DumpRelay1_FailtoClose := TRUE;
			Trips_DB.Section[j].Peak.DumpRly1FaultDelay_TON (IN:= FALSE);
		END_IF;
	ELSE
		Trips_DB.Section[j].Peak.DumpRly1FaultDelay_TON (IN:= FALSE);
	END_IF;

	//Peak dump rly2
		//fail to open
	IF LCP.Section[j].Peak.OpenDumpRelay2 = TRUE AND LCP.Section[j].Peak.DumpRelay2_close = TRUE THEN 
		//start timer
		Trips_DB.Section[j].Peak.DumpRly2FaultDelay_TON (IN := TRUE, PT := DumpRlyFaultDelay_PT); 
		
		IF Trips_DB.Section[j].Peak.DumpRly2FaultDelay_TON.Q = TRUE THEN 
			Trips_DB.Section[j].Peak.DumpRelay2_FailtoOpen := TRUE; 
			Trips_DB.Section[j].Peak.DumpRly2FaultDelay_TON (IN:= FALSE);
		END_IF;
	ELSE
		Trips_DB.Section[j].Peak.DumpRly2FaultDelay_TON (IN:= FALSE);
	END_IF;

		//fail to close
	IF LCP.Section[j].Peak.OpenDumpRelay2 = FALSE AND LCP.Section[j].Peak.DumpRelay2_close = FALSE THEN 
		//start timer
		Trips_DB.Section[j].Peak.DumpRly2FaultDelay_TON (IN := TRUE, PT := DumpRlyFaultDelay_PT); 
		IF Trips_DB.Section[j].Peak.DumpRly2FaultDelay_TON.Q = TRUE THEN 
			Trips_DB.Section[j].Peak.DumpRelay2_FailtoClose := TRUE; 
			
		END_IF;
	ELSE
		Trips_DB.Section[j].Peak.DumpRly2FaultDelay_TON (IN:= FALSE);
	END_IF;
//*************************************************************************************************

//Sust Charge rly1
		//fail to close
	IF LCP.Section[j].Sust.CloseChargeRelay1 = TRUE AND LCP.Section[j].Sust.ChargeRelay1_close = FALSE THEN 
		//start timer
		Trips_DB.Section[j].Sust.ChrgRly1FaultDelay_TON (IN:= TRUE, PT := ChrgRlyFaultDelay_PT);
		
